FUNCTION_BLOCK "FB_ShuttleInt"   // FB57, SCL
{ S7_Optimized_Access := 'TRUE' }
// stored: MemoryReserve 100, SetENOAutomatically false
   VAR_INPUT
      iStartSeqCond : Bool;   // Start Sequence Conditions
      iJobReq : Bool;   // Job Request - From Main
      iIntGateOpened : Bool;   // Internal Gate Opened - From DI
      iIntGateClosed : Bool;   // Internal Gate Closed - From DI
      iExtGateOpened : Bool;   // External Gate Opened - From DI
      iExtGateClosed : Bool;   // External Gate Closed - From DI
      iShuttlePosInt : Bool;   // Shuttle Inside the Machine - Param
      iShuttlePosSas : Bool;   // Shuttle Inside the Sas - Param
      iShuttlePosExt : Bool;   // Shuttle Outside the Machine - Param
      iShuttlePosIntSetPoint : LReal;   // Shuttle Outside Position Setpoint - Param
      iShuttlePosSasSetPoint : LReal;   // Shuttle SasPosition Setpoint - Param
      iShuttleMoving : Bool;   // Shuttle is moving - From FB_LoaderAxis
      iShuttleInPos : Bool;   // Shuttle pos. reached - From FB_LoaderAxis
      iIntLoaderInSafePos : Bool;   // Gripper in Safe Position - Param
      iPLC_DateAndTime : DTL;
      iStepPause : Bool;
   END_VAR
   VAR_OUTPUT
      oExtGateOpenReq { ExternalAccessible := 'False'; ExternalVisible := 'False'; ExternalWritable := 'False'} : Bool;   // External Gate Opening Request - To DO
      oExtGateCloseReq { ExternalAccessible := 'False'; ExternalVisible := 'False'; ExternalWritable := 'False'} : Bool;   // External Gate Closing Request - To DO
      oIntGateOpenReq { ExternalAccessible := 'False'; ExternalVisible := 'False'; ExternalWritable := 'False'} : Bool;   // Internal Gate Opening Request - To DO
      oIntGateCloseReq { ExternalAccessible := 'False'; ExternalVisible := 'False'; ExternalWritable := 'False'} : Bool;   // Internal Gate Closing Request - To DO
      oShuttleStartReq { ExternalAccessible := 'False'; ExternalVisible := 'False'; ExternalWritable := 'False'} : Bool;   // Shuttle Start Order - To FB_LoaderAxis
      oShuttlePosSetPoint { ExternalAccessible := 'False'; ExternalVisible := 'False'; ExternalWritable := 'False'} : Real;   // Shuttle Position Setpoint - To FB_LoaderAxis
   END_VAR
   VAR
      sCurrent_Step_NB : Int;   // Active Step Number
      sCheck_Step_Condition : Bool;   // Check Step Condition
      sOneStepForward : Bool;
      sRTOneStepForward : R_TRIG;
      sOneStepMode { S7_SetPoint := 'True'} : Bool;
      sStepForward : Bool;
      sInterface : "UDT_SequenceInterface";   // Sequence Interface
      sExtGateOpenReq { ExternalAccessible := 'False'; ExternalVisible := 'False'; ExternalWritable := 'False'} : Bool;   // External Gate Opening Request
      sExtGateCloseReq { ExternalAccessible := 'False'; ExternalVisible := 'False'; ExternalWritable := 'False'} : Bool;   // External Gate Closing Request
      sIntGateOpenReq { ExternalAccessible := 'False'; ExternalVisible := 'False'; ExternalWritable := 'False'} : Bool;   // Internal Gate Opening Request
      sIntGateCloseReq { ExternalAccessible := 'False'; ExternalVisible := 'False'; ExternalWritable := 'False'} : Bool;   // Internal Gate Closing Request
      sShuttleStartReq { ExternalAccessible := 'False'; ExternalVisible := 'False'; ExternalWritable := 'False'} : Bool;   // Shuttle Start Request
      sShuttlePosSetPoint { ExternalAccessible := 'False'; ExternalVisible := 'False'; ExternalWritable := 'False'} : Real;   // Shuttle Position Setpoint
      sHistory : Struct
         Activation : Bool;
         Steps : Array[0..99] of Int;
         Date_Time : Array[0..99] of DTL;
      END_STRUCT;
      StepText : "FB_GetTextErrorCode";
   END_VAR
   VAR_TEMP
      tIndex : Int;   // Index
   END_VAR
   VAR CONSTANT
      S00_INIT : Int := 0;
      S10_CHECK_SHUTTLE_POSITION : Int := 10;
      S20_CLOSE_INT_GATE : Int := 20;
      S30_OPEN_EXT_GATE : Int := 30;
      S40_SHUTTLE_TO_SAS_START_REQ : Int := 40;
      S50_SHUTTLE_TO_SAS_POS_REACHED : Int := 50;
      S60_CLOSE_EXT_GATE : Int := 60;
      S70_OPEN_INT_GATE : Int := 70;
      S80_MOVE_SHUTTLE_TO_IN_START_REQ : Int := 80;
      S90_MOVE_SHUTTLE_TO_IN_POS_REACHED : Int := 90;
      S100_CLOSE_INT_GATE : Int := 100;
      S195_JOB_DONE : Int := 195;
   END_VAR
   // StepText.sCode_error[0].ErrorCode := 0;
   // StepText.sCode_error[1].ErrorCode := 10;
   // StepText.sCode_error[2].ErrorCode := 20;
   // StepText.sCode_error[3].ErrorCode := 30;
   // StepText.sCode_error[4].ErrorCode := 40;
   // StepText.sCode_error[5].ErrorCode := 50;
   // StepText.sCode_error[6].ErrorCode := 60;
   // StepText.sCode_error[7].ErrorCode := 70;
   // StepText.sCode_error[8].ErrorCode := 80;
   // StepText.sCode_error[9].ErrorCode := 90;
   // StepText.sCode_error[10].ErrorCode := 95;
   // StepText.sCode_error[0].ErrorText := 'S00 : INIT';
   // StepText.sCode_error[1].ErrorText := 'S10 : CHECK SHUTTLE POSITION';
   // StepText.sCode_error[2].ErrorText := 'S20 : OPEN EXT GATE';
   // StepText.sCode_error[3].ErrorText := 'S30 : SHUTTLE TO SAS START REQ';
   // StepText.sCode_error[4].ErrorText := 'S40 : SHUTTLE TO SAS POS REACHED';
   // StepText.sCode_error[5].ErrorText := 'S50 : CLOSE EXT GATE';
   // StepText.sCode_error[6].ErrorText := 'S60 : OPEN INT GATE';
   // StepText.sCode_error[7].ErrorText := 'S70 : MOVE SHUTTLE TO IN START REQ';
   // StepText.sCode_error[8].ErrorText := 'S80 : MOVE SHUTTLE TO IN POS REACHED';
   // StepText.sCode_error[9].ErrorText := 'S90 : CLOSE INT GATE';
   // StepText.sCode_error[10].ErrorText := 'S95 : JOB DONE';
BEGIN
   REGION Description header 
       //==================================================================================
       // POSALUX Swiss SA / (C) Copyright 2025
       //----------------------------------------------------------------------------------
       // Title: FB_ShuttleInt
       // Comment/Function: 
       // Author: Fabien WALDT
       // Engineering: TIA Portal v17
       //----------------------------------------------------------------------------------
       // Change log table:
       // Version  | Date     | Expert in charge | Changes applied
       // ---------|----------|------------------|-----------------------------------------
       // 00.00.01 | 20250527 | WFA              | First released version
       // =================================================================================
   END_REGION

   REGION Define condition to start
       IF #iStartSeqCond THEN
           #sInterface.SequenceReleased := TRUE;
       ELSE
           // Standard sequencer controls
           #sInterface.SequenceReleased := FALSE;
           #sCurrent_Step_NB := #S00_INIT;
           #sInterface.SequenceRun := FALSE;
           #sInterface.JobDone := FALSE;
           #sCheck_Step_Condition := FALSE;

           // Dedicated sequencer controls
           #sExtGateOpenReq := FALSE;
           #sExtGateCloseReq := FALSE;
           #sIntGateOpenReq := FALSE;
           #sIntGateCloseReq := FALSE;
           #sShuttleStartReq := FALSE;
           #sShuttlePosSetPoint := 0.0;
           // Add specifics controls 
       END_IF;

       // Reset interface error
       IF #sInterface.Reset THEN
           #sInterface.Error := FALSE;
       END_IF;

       // Reset start when axis in position
       IF #iShuttleInPos THEN
           #sShuttleStartReq := FALSE;
       END_IF;

       // One step forward
       #sRTOneStepForward.CLK := #sOneStepForward;
       #sRTOneStepForward();
       #sStepForward := (NOT #sOneStepMode OR (#sOneStepMode AND #sRTOneStepForward.Q)) AND NOT #iStepPause;
       #sOneStepForward := FALSE;
   END_REGION

   REGION Sequence Function
       CASE #sCurrent_Step_NB OF
           #S00_INIT:
               REGION S00 INIT
                   #sCheck_Step_Condition := TRUE;
               END_REGION
           #S10_CHECK_SHUTTLE_POSITION:
               REGION S10_CHECK_SHUTTLE_POSITION
                   #sCheck_Step_Condition := TRUE;
               END_REGION
           #S20_CLOSE_INT_GATE:
               REGION S20_CLOSE_INT_GATE
                   #sIntGateOpenReq := FALSE;
                   #sIntGateCloseReq := TRUE;
                   #sCheck_Step_Condition := TRUE;
               END_REGION
           #S30_OPEN_EXT_GATE:
               REGION S30_OPEN_EXT_GATE
                   #sExtGateOpenReq := TRUE;
                   #sExtGateCloseReq := FALSE;
                   #sCheck_Step_Condition := TRUE;
               END_REGION
           #S40_SHUTTLE_TO_SAS_START_REQ:
               REGION S40_SHUTTLE_TO_SAS_START_REQ
                   #sShuttleStartReq := #iExtGateOpened AND NOT #iShuttlePosSas;
                   #sShuttlePosSetPoint := LREAL_TO_REAL(#iShuttlePosSasSetPoint);
                   #sCheck_Step_Condition := TRUE;
               END_REGION
           #S50_SHUTTLE_TO_SAS_POS_REACHED:
               REGION S50_SHUTTLE_TO_SAS_POS_REACHED
                   #sCheck_Step_Condition := TRUE;
               END_REGION
           #S60_CLOSE_EXT_GATE:
               REGION S60_CLOSE_EXT_GATE
                   #sExtGateOpenReq := FALSE;
                   #sExtGateCloseReq := TRUE;
                   #sCheck_Step_Condition := TRUE;
               END_REGION
           #S70_OPEN_INT_GATE:
               REGION S70_OPEN_INT_GATE
                   #sIntGateOpenReq := TRUE;
                   #sIntGateCloseReq := FALSE;
                   #sCheck_Step_Condition := TRUE;
               END_REGION
           #S80_MOVE_SHUTTLE_TO_IN_START_REQ:
               REGION S80_MOVE_SHUTTLE_TO_IN_START_REQ
                   #sShuttleStartReq := #iIntGateOpened AND NOT #iShuttlePosInt;
                   #sShuttlePosSetPoint := LREAL_TO_REAL(#iShuttlePosIntSetPoint);
                   #sCheck_Step_Condition := TRUE;
               END_REGION
           #S90_MOVE_SHUTTLE_TO_IN_POS_REACHED:
               REGION S90_MOVE_SHUTTLE_TO_IN_POS_REACHED
                   #sCheck_Step_Condition := TRUE;
               END_REGION
           #S100_CLOSE_INT_GATE:
               REGION S100_CLOSE_INT_GATE
                   #sIntGateOpenReq := FALSE;
                   #sIntGateCloseReq := TRUE;
                   #sExtGateOpenReq := FALSE;
                   #sExtGateCloseReq := TRUE;
                   #sCheck_Step_Condition := TRUE;
               END_REGION
           #S195_JOB_DONE:
               REGION S195_JOB_DONE
                   #sInterface.JobDone := TRUE;
                   #sCheck_Step_Condition := TRUE;
               END_REGION
           ELSE:
               #sInterface.Error := TRUE;
       END_CASE;
   END_REGION

   REGION Sequence Next Step Condition
       IF #sCheck_Step_Condition THEN
           CASE #sCurrent_Step_NB OF
               #S00_INIT:
                   REGION S00 INIT
                       IF #sInterface.SequenceReleased AND #iJobReq THEN
                           #sCurrent_Step_NB := #S10_CHECK_SHUTTLE_POSITION;
                           #sInterface.SequenceRun := TRUE;
                           #sCheck_Step_Condition := FALSE;
                       ELSE
                           #sInterface.SequenceRun := FALSE;
                       END_IF;
                   END_REGION
               #S10_CHECK_SHUTTLE_POSITION:
                   REGION S10_CHECK_SHUTTLE_POSITION
                       IF #sInterface.SequenceReleased AND #sStepForward AND #iShuttlePosExt THEN
                           #sCurrent_Step_NB := #S20_CLOSE_INT_GATE;
                           #sCheck_Step_Condition := FALSE;
                       ELSIF #sInterface.SequenceReleased AND #sStepForward AND #iShuttlePosSas THEN
                           #sCurrent_Step_NB := #S60_CLOSE_EXT_GATE;
                           #sCheck_Step_Condition := FALSE;
                       ELSIF #sInterface.SequenceReleased AND #sStepForward AND #iShuttlePosInt THEN
                           #sCurrent_Step_NB := #S100_CLOSE_INT_GATE;
                           #sCheck_Step_Condition := FALSE;
                       END_IF;
                   END_REGION
               #S20_CLOSE_INT_GATE:
                   REGION S20_CLOSE_INT_GATE
                       IF #sInterface.SequenceReleased AND #sStepForward AND #iIntGateClosed THEN
                           #sCurrent_Step_NB := #S30_OPEN_EXT_GATE;
                           #sCheck_Step_Condition := FALSE;
                       END_IF;
                   END_REGION
               #S30_OPEN_EXT_GATE:
                   REGION S30_OPEN_EXT_GATE
                       IF #sInterface.SequenceReleased AND #sStepForward AND #iExtGateOpened THEN
                           #sCurrent_Step_NB := #S40_SHUTTLE_TO_SAS_START_REQ;
                           #sCheck_Step_Condition := FALSE;
                       END_IF;
                   END_REGION
               #S40_SHUTTLE_TO_SAS_START_REQ:
                   REGION S40_SHUTTLE_TO_SAS_START_REQ
                      // IF #sInterface.SequenceReleased AND #sStepForward AND (#ShuttleMoving OR #ShuttlePosSas)  THEN
                       IF #sInterface.SequenceReleased AND (#iShuttleMoving OR #iShuttlePosSas)  THEN
                           #sCurrent_Step_NB := #S50_SHUTTLE_TO_SAS_POS_REACHED;
                           #sCheck_Step_Condition := FALSE;
                       END_IF;
                   END_REGION
               #S50_SHUTTLE_TO_SAS_POS_REACHED:
                   REGION S50_SHUTTLE_TO_SAS_POS_REACHED
                       IF #sInterface.SequenceReleased AND #sStepForward AND NOT #sShuttleStartReq AND #iShuttlePosSas THEN
                           #sCurrent_Step_NB := #S60_CLOSE_EXT_GATE;
                           #sCheck_Step_Condition := FALSE;
                       END_IF;
                   END_REGION
               #S60_CLOSE_EXT_GATE:
                   REGION S60_CLOSE_EXT_GATE
                       IF #sInterface.SequenceReleased AND #sStepForward AND #iExtGateClosed THEN
                           #sCurrent_Step_NB := #S70_OPEN_INT_GATE;
                           #sCheck_Step_Condition := FALSE;
                       END_IF;
                   END_REGION
               #S70_OPEN_INT_GATE:
                   REGION S70_OPEN_INT_GATE
                       IF #sInterface.SequenceReleased AND #sStepForward AND #iIntGateOpened THEN
                           #sCurrent_Step_NB := #S80_MOVE_SHUTTLE_TO_IN_START_REQ;
                           #sCheck_Step_Condition := FALSE;
                       END_IF;
                   END_REGION
               #S80_MOVE_SHUTTLE_TO_IN_START_REQ:
                   REGION S80_MOVE_SHUTTLE_TO_IN_START_REQ
                       IF #sInterface.SequenceReleased AND (#iShuttleMoving OR #iShuttlePosInt) THEN
                           #sCurrent_Step_NB := #S90_MOVE_SHUTTLE_TO_IN_POS_REACHED;
                           #sCheck_Step_Condition := FALSE;
                       END_IF;
                   END_REGION
               #S90_MOVE_SHUTTLE_TO_IN_POS_REACHED:
                   REGION S90_MOVE_SHUTTLE_TO_IN_POS_REACHED
                       IF #sInterface.SequenceReleased AND #sStepForward AND NOT #sShuttleStartReq AND #iShuttlePosInt THEN
                           #sCurrent_Step_NB := #S100_CLOSE_INT_GATE;
                           #sCheck_Step_Condition := FALSE;
                       END_IF;
                   END_REGION
               #S100_CLOSE_INT_GATE:
                   REGION S100_CLOSE_INT_GATE
                       IF #sInterface.SequenceReleased AND #sStepForward AND #iIntGateClosed AND #iExtGateClosed THEN
                           #sCurrent_Step_NB := #S195_JOB_DONE;
                           #sCheck_Step_Condition := FALSE;
                       END_IF;
                   END_REGION
               #S195_JOB_DONE:
                   REGION S195_JOB_DONE
                       IF NOT #iJobReq THEN
                           #sCurrent_Step_NB := #S00_INIT;
                           #sCheck_Step_Condition := FALSE;
                           #sInterface.JobDone := FALSE;
                       END_IF;
                   END_REGION
               ELSE
                   #sInterface.Error := TRUE;
           END_CASE;
       END_IF;
   END_REGION

   REGION Outputs Update
       #oExtGateOpenReq  := #sExtGateOpenReq;
       #oExtGateCloseReq := #sExtGateCloseReq;
       #oIntGateOpenReq  := #sIntGateOpenReq;
       #oIntGateCloseReq := #sIntGateCloseReq;
       #oShuttleStartReq := #sShuttleStartReq AND ((#iShuttlePosInt AND #iIntLoaderInSafePos) OR NOT #iShuttlePosInt);
       #oShuttlePosSetPoint:= #sShuttlePosSetPoint;
   END_REGION

   REGION Steps - Date and Time History
       IF #sHistory.Activation THEN
           IF #sHistory.Steps[0] <> #sCurrent_Step_NB THEN
               FOR #tIndex := 98 TO 0 BY -1 DO
                   #sHistory.Steps[#tIndex + 1] := #sHistory.Steps[#tIndex];
                   #sHistory.Date_Time[#tIndex + 1] := #sHistory.Date_Time[#tIndex];
               END_FOR;
               #sHistory.Steps[0] := #sCurrent_Step_NB;
               #sHistory.Date_Time[0] := #iPLC_DateAndTime;
           END_IF;
       END_IF;
   END_REGION

   REGION Steps Text
       #StepText(iErrorCode:=#sCurrent_Step_NB,
                 oErrorText=>#StepText.oErrorText);
   END_REGION
END_FUNCTION_BLOCK

FUNCTION_BLOCK "FB_ShuttleExt"   // FB59, SCL
{ S7_Optimized_Access := 'TRUE' }
// stored: MemoryReserve 100, SetENOAutomatically false
   VAR_INPUT
      iStartSeqCond : Bool;   // Start Sequence Conditions
      iJobReq : Bool;   // Job Request - From Main
      iIntGateOpened : Bool;   // Internal Gate Opened - From DI
      iIntGateClosed : Bool;   // Internal Gate Closed - From DI
      iExtGateOpened : Bool;   // External Gate Opened - From DI
      iExtGateClosed : Bool;   // External Gate Closed - From DI
      iShuttlePosInt : Bool;   // Shuttle Inside the Machine - Param
      iShuttlePosSas : Bool;   // Shuttle Inside the Sas - Param
      iShuttlePosExt : Bool;   // Shuttle Outside the Machine - Param
      iShuttlePosExtSetPoint : LReal;   // Shuttle Outside Position Setpoint - Param
      iShuttlePosSasSetPoint : LReal;   // Shuttle SasPosition Setpoint - Param
      iShuttleMoving : Bool;   // Shuttle is moving - From FB_LoaderAxis
      iShuttleInPos : Bool;   // Shuttle pos. reached - From FB_LoaderAxis
      iExtLoaderInSafePos : Bool;   // Gripper in Safe Position - Param
      iPLC_DateAndTime : DTL;
      iStepPause : Bool;
   END_VAR
   VAR_OUTPUT
      oExtGateOpenReq { ExternalAccessible := 'False'; ExternalVisible := 'False'; ExternalWritable := 'False'} : Bool;   // External Gate Opening Request - To DO
      oExtGateCloseReq { ExternalAccessible := 'False'; ExternalVisible := 'False'; ExternalWritable := 'False'} : Bool;   // External Gate Closing Request - To DO
      oIntGateOpenReq { ExternalAccessible := 'False'; ExternalVisible := 'False'; ExternalWritable := 'False'} : Bool;   // Internal Gate Opening Request - To DO
      oIntGateCloseReq { ExternalAccessible := 'False'; ExternalVisible := 'False'; ExternalWritable := 'False'} : Bool;   // Internal Gate Closing Request - To DO
      oShuttleStartReq { ExternalAccessible := 'False'; ExternalVisible := 'False'; ExternalWritable := 'False'} : Bool;   // Shuttle Start Order - To FB_LoaderAxis
      oShuttlePosSetPoint { ExternalAccessible := 'False'; ExternalVisible := 'False'; ExternalWritable := 'False'} : Real;   // Shuttle Position Setpoint - To FB_LoaderAxis
   END_VAR
   VAR
      sCurrent_Step_NB : Int;   // Active Step Number
      sCheck_Step_Condition : Bool;   // Check Step Condition
      sOneStepForward : Bool;
      sRTOneStepForward : R_TRIG;
      sOneStepMode { S7_SetPoint := 'True'} : Bool;
      sStepForward : Bool;
      sInterface : "UDT_SequenceInterface";   // Sequence Interface
      sExtGateOpenReq { ExternalAccessible := 'False'; ExternalVisible := 'False'; ExternalWritable := 'False'} : Bool;   // External Gate Opening Request
      sExtGateCloseReq { ExternalAccessible := 'False'; ExternalVisible := 'False'; ExternalWritable := 'False'} : Bool;   // External Gate Closing Request
      sIntGateOpenReq { ExternalAccessible := 'False'; ExternalVisible := 'False'; ExternalWritable := 'False'} : Bool;   // Internal Gate Opening Request
      sIntGateCloseReq { ExternalAccessible := 'False'; ExternalVisible := 'False'; ExternalWritable := 'False'} : Bool;   // Internal Gate Closing Request
      sShuttleStartReq { ExternalAccessible := 'False'; ExternalVisible := 'False'; ExternalWritable := 'False'} : Bool;   // Shuttle Start Request
      sShuttlePosSetPoint { ExternalAccessible := 'False'; ExternalVisible := 'False'; ExternalWritable := 'False'} : Real;   // Shuttle Position Setpoint
      sHistory : Struct
         Activation : Bool;
         Steps : Array[0..99] of Int;
         Date_Time : Array[0..99] of DTL;
      END_STRUCT;
      StepText : "FB_GetTextErrorCode";
   END_VAR
   VAR_TEMP
      tIndex : Int;   // Index
   END_VAR
   VAR CONSTANT
      S00_INIT : Int := 0;
      S10_CHECK_SHUTTLE_POSITION : Int := 10;
      S20_CLOSE_EXT_GATE : Int := 20;
      S30_OPEN_INT_GATE : Int := 30;
      S40_SHUTTLE_TO_SAS_START_REQ : Int := 40;
      S50_SHUTTLE_TO_SAS_POS_REACHED : Int := 50;
      S60_CLOSE_INT_GATE : Int := 60;
      S70_OPEN_EXT_GATE : Int := 70;
      S80_MOVE_SHUTTLE_TO_OUT_START_REQ : Int := 80;
      S90_MOVE_SHUTTLE_TO_OUT_POS_REACHED : Int := 90;
      S100_CLOSE_EXT_GATE : Int := 100;
      S195_JOB_DONE : Int := 195;
   END_VAR
   // StepText.sCode_error[0].ErrorCode := 0;
   // StepText.sCode_error[1].ErrorCode := 10;
   // StepText.sCode_error[2].ErrorCode := 20;
   // StepText.sCode_error[3].ErrorCode := 30;
   // StepText.sCode_error[4].ErrorCode := 40;
   // StepText.sCode_error[5].ErrorCode := 50;
   // StepText.sCode_error[6].ErrorCode := 60;
   // StepText.sCode_error[7].ErrorCode := 70;
   // StepText.sCode_error[8].ErrorCode := 80;
   // StepText.sCode_error[9].ErrorCode := 90;
   // StepText.sCode_error[10].ErrorCode := 95;
   // StepText.sCode_error[0].ErrorText := 'S00 : INIT';
   // StepText.sCode_error[1].ErrorText := 'S10 : CHECK SHUTTLE POSITION';
   // StepText.sCode_error[2].ErrorText := 'S20 : OPEN INT GATE';
   // StepText.sCode_error[3].ErrorText := 'S30 : SHUTTLE TO SAS START REQ';
   // StepText.sCode_error[4].ErrorText := 'S40 : SHUTTLE TO SAS POS REACHED';
   // StepText.sCode_error[5].ErrorText := 'S50 : CLOSE INT GATE';
   // StepText.sCode_error[6].ErrorText := 'S60 : OPEN EXT GATE';
   // StepText.sCode_error[7].ErrorText := 'S70 : MOVE SHUTTLE TO OUT START REQ';
   // StepText.sCode_error[8].ErrorText := 'S80 : MOVE SHUTTLE TO OUT POS REACHED';
   // StepText.sCode_error[9].ErrorText := 'S90 : CLOSE EXT GATE';
   // StepText.sCode_error[10].ErrorText := 'S95 : JOB DONE';
BEGIN
   REGION Description header 
       //==================================================================================
       // POSALUX Swiss SA / (C) Copyright 2025
       //----------------------------------------------------------------------------------
       // Title: FB_ShuttleExt
       // Comment/Function: 
       // Author: Fabien WALDT
       // Engineering: TIA Portal v17
       //----------------------------------------------------------------------------------
       // Change log table:
       // Version  | Date     | Expert in charge | Changes applied
       // ---------|----------|------------------|-----------------------------------------
       // 00.00.01 | 20250527 | WFA              | First released version
       // =================================================================================
   END_REGION

   REGION Define condition to start
       IF #iStartSeqCond THEN
           #sInterface.SequenceReleased := TRUE;
       ELSE
           // Standard sequencer controls
           #sInterface.SequenceReleased := FALSE;
           #sCurrent_Step_NB := #S00_INIT;
           #sInterface.SequenceRun := FALSE;
           #sInterface.JobDone := FALSE;
           #sCheck_Step_Condition := FALSE;

           // Dedicated sequencer controls
           #sExtGateOpenReq := FALSE;
           #sExtGateCloseReq := FALSE;
           #sIntGateOpenReq := FALSE;
           #sIntGateCloseReq := FALSE;
           #sShuttleStartReq := FALSE;
           #sShuttlePosSetPoint := 0.0;
           // Add specifics controls 
       END_IF;

       // Reset interface error
       IF #sInterface.Reset THEN
           #sInterface.Error := FALSE;
       END_IF;

       // Reset start when axis in position
       IF #iShuttleInPos THEN
           #sShuttleStartReq := FALSE;
       END_IF;

       // One step forward
       #sRTOneStepForward.CLK := #sOneStepForward;
       #sRTOneStepForward();
       #sStepForward := (NOT #sOneStepMode OR (#sOneStepMode AND #sRTOneStepForward.Q)) AND NOT #iStepPause;
       #sOneStepForward := FALSE;
   END_REGION

   REGION Sequence Function
       CASE #sCurrent_Step_NB OF
           #S00_INIT:
               REGION S00 INIT
                   #sCheck_Step_Condition := TRUE;
               END_REGION
           #S10_CHECK_SHUTTLE_POSITION:
               REGION S10_CHECK_SHUTTLE_POSITION
                   #sCheck_Step_Condition := TRUE;
               END_REGION
           #S20_CLOSE_EXT_GATE:
               REGION S20_CLOSE_EXT_GATE
                   #sExtGateOpenReq := FALSE;
                   #sExtGateCloseReq := TRUE;
                   #sCheck_Step_Condition := TRUE;
               END_REGION
           #S30_OPEN_INT_GATE:
               REGION S30_OPEN_INT_GATE
                   #sIntGateOpenReq := TRUE;
                   #sIntGateCloseReq := FALSE;
                   #sCheck_Step_Condition := TRUE;
               END_REGION
           #S40_SHUTTLE_TO_SAS_START_REQ:
               REGION S40_SHUTTLE_TO_SAS_START_REQ
                   #sShuttleStartReq := #iIntGateOpened AND NOT #iShuttlePosSas;
                   #sShuttlePosSetPoint := LREAL_TO_REAL(#iShuttlePosSasSetPoint);
                   #sCheck_Step_Condition := TRUE;
               END_REGION
           #S50_SHUTTLE_TO_SAS_POS_REACHED:
               REGION S50_SHUTTLE_TO_SAS_POS_REACHED
                   #sCheck_Step_Condition := TRUE;
               END_REGION
           #S60_CLOSE_INT_GATE:
               REGION S60_CLOSE_INT_GATE
                   #sIntGateOpenReq := FALSE;
                   #sIntGateCloseReq := TRUE;
                   #sCheck_Step_Condition := TRUE;
               END_REGION
           #S70_OPEN_EXT_GATE:
               REGION S70_OPEN_EXT_GATE
                   #sExtGateOpenReq := TRUE;
                   #sExtGateCloseReq := FALSE;
                   #sCheck_Step_Condition := TRUE;
               END_REGION
           #S80_MOVE_SHUTTLE_TO_OUT_START_REQ:
               REGION S80_MOVE_SHUTTLE_TO_OUT_START_REQ
                   #sShuttleStartReq := #iExtGateOpened AND NOT #iShuttlePosExt;
                   #sShuttlePosSetPoint := LREAL_TO_REAL(#iShuttlePosExtSetPoint);
                   #sCheck_Step_Condition := TRUE;
               END_REGION
           #S90_MOVE_SHUTTLE_TO_OUT_POS_REACHED:
               REGION S90_MOVE_SHUTTLE_TO_OUT_POS_REACHED
                   #sCheck_Step_Condition := TRUE;
               END_REGION
           #S100_CLOSE_EXT_GATE:
               REGION S100_CLOSE_EXT_GATE
                   #sIntGateOpenReq := FALSE;
                   #sIntGateCloseReq := TRUE;
                   #sExtGateOpenReq := FALSE;
                   #sExtGateCloseReq := TRUE;
                   #sCheck_Step_Condition := TRUE;
               END_REGION
           #S195_JOB_DONE:
               REGION S195_JOB_DONE
                   #sInterface.JobDone := TRUE;
                   #sCheck_Step_Condition := TRUE;
               END_REGION
           ELSE:
               #sInterface.Error := TRUE;
       END_CASE;
   END_REGION

   REGION Sequence Next Step Condition
       IF #sCheck_Step_Condition THEN
           CASE #sCurrent_Step_NB OF
               #S00_INIT:
                   REGION S00 INIT
                       IF #sInterface.SequenceReleased AND #iJobReq THEN
                           #sCurrent_Step_NB := #S10_CHECK_SHUTTLE_POSITION;
                           #sInterface.SequenceRun := TRUE;
                           #sCheck_Step_Condition := FALSE;
                       ELSE
                           #sInterface.SequenceRun := FALSE;
                       END_IF;
                   END_REGION
               #S10_CHECK_SHUTTLE_POSITION:
                   REGION S10_CHECK_SHUTTLE_POSITION
                       IF #sInterface.SequenceReleased AND #sStepForward AND #iShuttlePosInt THEN
                           #sCurrent_Step_NB := #S20_CLOSE_EXT_GATE;
                           #sCheck_Step_Condition := FALSE;
                       ELSIF #sInterface.SequenceReleased AND #sStepForward AND #iShuttlePosSas THEN
                           #sCurrent_Step_NB := #S60_CLOSE_INT_GATE;
                           #sCheck_Step_Condition := FALSE;
                       ELSIF #sInterface.SequenceReleased AND #sStepForward AND #iShuttlePosExt THEN
                           #sCurrent_Step_NB := #S100_CLOSE_EXT_GATE;
                           #sCheck_Step_Condition := FALSE;
                       END_IF;
                   END_REGION
               #S20_CLOSE_EXT_GATE:
                   REGION S20_CLOSE_EXT_GATE
                       IF #sInterface.SequenceReleased AND #sStepForward AND #iExtGateClosed THEN
                           #sCurrent_Step_NB := #S30_OPEN_INT_GATE;
                           #sCheck_Step_Condition := FALSE;
                       END_IF;
                   END_REGION
               #S30_OPEN_INT_GATE:
                   REGION S30_OPEN_INT_GATE
                       IF #sInterface.SequenceReleased AND #sStepForward AND #iIntGateOpened THEN
                           #sCurrent_Step_NB := #S40_SHUTTLE_TO_SAS_START_REQ;
                           #sCheck_Step_Condition := FALSE;
                       END_IF;
                   END_REGION
               #S40_SHUTTLE_TO_SAS_START_REQ:
                   REGION S40_SHUTTLE_TO_SAS_START_REQ
                     //  IF #sInterface.SequenceReleased AND #sStepForward AND (#ShuttleMoving OR #ShuttlePosSas) THEN
                       IF #sInterface.SequenceReleased AND (#iShuttleMoving OR #iShuttlePosSas) THEN
                           #sCurrent_Step_NB := #S50_SHUTTLE_TO_SAS_POS_REACHED;
                           #sCheck_Step_Condition := FALSE;
                       END_IF;
                   END_REGION
               #S50_SHUTTLE_TO_SAS_POS_REACHED:
                   REGION S50_SHUTTLE_TO_SAS_POS_REACHED
                       IF #sInterface.SequenceReleased AND #sStepForward AND NOT #sShuttleStartReq AND #iShuttlePosSas THEN
                           #sCurrent_Step_NB := #S60_CLOSE_INT_GATE;
                           #sCheck_Step_Condition := FALSE;
                       END_IF;
                   END_REGION
               #S60_CLOSE_INT_GATE:
                   REGION S60_CLOSE_INT_GATE
                       IF #sInterface.SequenceReleased AND #sStepForward AND #iIntGateClosed THEN
                           #sCurrent_Step_NB := #S70_OPEN_EXT_GATE;
                           #sCheck_Step_Condition := FALSE;
                       END_IF;
                   END_REGION
               #S70_OPEN_EXT_GATE:
                   REGION S70_OPEN_EXT_GATE
                       IF #sInterface.SequenceReleased AND #sStepForward AND #iExtGateOpened THEN
                           #sCurrent_Step_NB := #S80_MOVE_SHUTTLE_TO_OUT_START_REQ;
                           #sCheck_Step_Condition := FALSE;
                       END_IF;
                   END_REGION
               #S80_MOVE_SHUTTLE_TO_OUT_START_REQ:
                   REGION S80_MOVE_SHUTTLE_TO_OUT_START_REQ
                       IF #sInterface.SequenceReleased AND (#iShuttleMoving OR #iShuttlePosExt) THEN
                           #sCurrent_Step_NB := #S90_MOVE_SHUTTLE_TO_OUT_POS_REACHED;
                           #sCheck_Step_Condition := FALSE;
                       END_IF;
                   END_REGION
               #S90_MOVE_SHUTTLE_TO_OUT_POS_REACHED:
                   REGION S90_MOVE_SHUTTLE_TO_OUT_POS_REACHED
                       IF #sInterface.SequenceReleased AND #sStepForward AND NOT #sShuttleStartReq AND #iShuttlePosExt THEN
                           #sCurrent_Step_NB := #S100_CLOSE_EXT_GATE;
                           #sCheck_Step_Condition := FALSE;
                       END_IF;
                   END_REGION
               #S100_CLOSE_EXT_GATE:
                   REGION S100_CLOSE_EXT_GATE
                       IF #sInterface.SequenceReleased AND #sStepForward AND #iIntGateClosed AND #iExtGateClosed THEN
                           #sCurrent_Step_NB := #S195_JOB_DONE;
                           #sCheck_Step_Condition := FALSE;
                       END_IF;
                   END_REGION
               #S195_JOB_DONE:
                   REGION S195_JOB_DONE
                       IF NOT #iJobReq THEN
                           #sCurrent_Step_NB := #S00_INIT;
                           #sCheck_Step_Condition := FALSE;
                           #sInterface.JobDone := FALSE;
                       END_IF;
                   END_REGION
               ELSE
                   #sInterface.Error := TRUE;
           END_CASE;
       END_IF;
   END_REGION

   REGION Outputs Update
       #oExtGateOpenReq  := #sExtGateOpenReq;
       #oExtGateCloseReq := #sExtGateCloseReq;
       #oIntGateOpenReq  := #sIntGateOpenReq;
       #oIntGateCloseReq := #sIntGateCloseReq;
       #oShuttleStartReq:= #sShuttleStartReq AND ((#iShuttlePosExt AND #iExtLoaderInSafePos) OR NOT #iShuttlePosExt);
       #oShuttlePosSetPoint:= #sShuttlePosSetPoint;
   END_REGION

   REGION Steps - Date and Time History
       IF #sHistory.Activation THEN
           IF #sHistory.Steps[0] <> #sCurrent_Step_NB THEN
               FOR #tIndex := 98 TO 0 BY -1 DO
                   #sHistory.Steps[#tIndex + 1] := #sHistory.Steps[#tIndex];
                   #sHistory.Date_Time[#tIndex + 1] := #sHistory.Date_Time[#tIndex];
               END_FOR;
               #sHistory.Steps[0] := #sCurrent_Step_NB;
               #sHistory.Date_Time[0] := #iPLC_DateAndTime;
           END_IF;
       END_IF;
   END_REGION

   REGION Steps Text
       #StepText(iErrorCode := #sCurrent_Step_NB,
                 oErrorText => #StepText.oErrorText);
   END_REGION
END_FUNCTION_BLOCK

FUNCTION_BLOCK "FB_ExtLoadUnload"   // FB61, SCL
{ S7_Optimized_Access := 'TRUE' }
// stored: MemoryReserve 100, SetENOAutomatically false
   VAR_INPUT
      iStartSeqCond : Bool;   // Start Sequence Conditions
      iJobReq : Bool;   // Job Request - From Main
      iShuttleExtLoadUnloadAutoPos : Bool;   // Load/Unload Auto Pos. Reached - Param
      iShuttleExtLoadUnloadAutoPosSetPoint : LReal;   // Load/Unload Auto Pos. Setpoint - Param
      iShuttleExtLoadUnloadManuPos : Bool;   // Load/Unload Manu Pos. Reached - Param
      iShuttleExtLoadUnloadManuPosSetPoint : LReal;   // Load/Unload Manu Pos. Setpoint - Param
      iShuttleMoving : Bool;   // Shuttle is moving - From FB_LoaderAxis
      iShuttleInPos : Bool;   // Shuttle pos. reached - From FB_LoaderAxis
      iCommunicationWithExtLoaderDone : Bool;   // Communication Done - From Ext Loader
      iLoadUnloadMsgManuModeAck : Bool;   // Load/Unload Message Ack - From HMI
      iAutoMode : Bool;
      iSemiAutoMode : Bool;
      iFillingMode : Bool;   // Filling Mode - From Machine States
      iEmptyingMode : Bool;   // Emptying Mode - From Machine States
      iPLC_DateAndTime : DTL;
      iStepPause : Bool;
   END_VAR
   VAR_OUTPUT
      oShuttleStartReq { ExternalAccessible := 'False'; ExternalVisible := 'False'; ExternalWritable := 'False'} : Bool;   // Shuttle Start Order - To FB_LoaderAxis
      oShuttlePosSetPoint { ExternalAccessible := 'False'; ExternalVisible := 'False'; ExternalWritable := 'False'} : Real;   // Shuttle Position Setpoint - To FB_LoaderAxis
      oStartCommunicationWithExtLoader : Bool;   // Start Communication - To Ext Loader
      oSetLoadUnloadMsgManuMode : Bool;   // Set Load/Unload Message - To HMI
   END_VAR
   VAR
      sCurrent_Step_NB : Int;   // Active Step Number
      sCheck_Step_Condition : Bool;
      sOneStepForward : Bool;
      sRTOneStepForward : R_TRIG;
      sOneStepMode { S7_SetPoint := 'True'} : Bool;
      sStepForward : Bool;
      sInterface : "UDT_SequenceInterface";
      sShuttleStartReq { ExternalAccessible := 'False'; ExternalVisible := 'False'; ExternalWritable := 'False'} : Bool;
      sShuttlePosSetPoint { ExternalAccessible := 'False'; ExternalVisible := 'False'; ExternalWritable := 'False'} : Real;
      sHistory : Struct
         Activation : Bool;
         Steps : Array[0..99] of Int;
         Date_Time : Array[0..99] of DTL;
      END_STRUCT;
      StepText : "FB_GetTextErrorCode";
   END_VAR
   VAR_TEMP
      tIndex : Int;   // Index
   END_VAR
   VAR CONSTANT
      S00_INIT : Int := 0;
      S10_CHECK_EXT_LOAD_UNLOAD_OPTION : Int := 10;
      S20_SHUTTLE_TO_EXT_LOAD_UNLOAD_POS_START_REQ : Int := 20;
      S30_SHUTTLE_TO_EXT_LOAD_UNLOAD_POS_REACHED : Int := 30;
      S40_SET_EXCHANGE_EXT_LOADER_LOAD_UNLOAD : Int := 40;
      S50_EXCHANGE_EXT_LOADER_IN_PROGRESS : Int := 50;
      S60_EXCHANGE_EXT_LOADER_ACQUIT : Int := 60;
      S70_SET_EXCHANGE_EXT_LOADER_UNLOAD : Int := 70;
      S80_EXCHANGE_EXT_LOADER_IN_PROGRESS : Int := 80;
      S90_EXCHANGE_EXT_LOADER_ACQUIT : Int := 90;
      S100_SET_EXCHANGE_EXT_LOADER_UNLOAD : Int := 100;
      S110_EXCHANGE_EXT_LOADER_IN_PROGRESS : Int := 110;
      S120_EXCHANGE_EXT_LOADER_ACQUIT : Int := 120;
      S130_SHUTTLE_TO_EXT_LOAD_UNLOAD_MANU_POS_START_REQ : Int := 130;
      S140_SHUTTLE_TO_EXT_LOAD_UNLOAD_MANU_POS_REACHED : Int := 140;
      S150_OPERATOR_MESSAGE : Int := 150;
      S195_JOB_DONE : Int := 195;
   END_VAR
   // StepText.sCode_error[0].ErrorCode := 0;
   // StepText.sCode_error[1].ErrorCode := 10;
   // StepText.sCode_error[2].ErrorCode := 20;
   // StepText.sCode_error[3].ErrorCode := 30;
   // StepText.sCode_error[4].ErrorCode := 40;
   // StepText.sCode_error[5].ErrorCode := 50;
   // StepText.sCode_error[6].ErrorCode := 60;
   // StepText.sCode_error[7].ErrorCode := 70;
   // StepText.sCode_error[8].ErrorCode := 80;
   // StepText.sCode_error[9].ErrorCode := 90;
   // StepText.sCode_error[10].ErrorCode := 95;
BEGIN
   REGION Description header 
       //==================================================================================
       // POSALUX Swiss SA / (C) Copyright 2025
       //----------------------------------------------------------------------------------
       // Title: FB_ExtLoadUnload
       // Comment/Function: 
       // Author: Fabien WALDT
       // Engineering: TIA Portal v17
       //----------------------------------------------------------------------------------
       // Change log table:
       // Version  | Date     | Expert in charge | Changes applied
       // ---------|----------|------------------|-----------------------------------------
       // 00.00.01 | 20250527 | WFA              | First released version
       // =================================================================================
   END_REGION

   REGION Define condition to start
       IF #iStartSeqCond THEN
           #sInterface.SequenceReleased := TRUE;
       ELSE
           // Standard sequencer controls
           #sInterface.SequenceReleased := FALSE;
           #sCurrent_Step_NB := #S00_INIT;
           #sInterface.SequenceRun := FALSE;
           #sInterface.JobDone := FALSE;
           #sCheck_Step_Condition := FALSE;

           // Dedicated sequencer controls
           #sShuttleStartReq := FALSE;
           #sShuttlePosSetPoint := 0.0;
           #oStartCommunicationWithExtLoader := FALSE;
           // Add specifics controls 
       END_IF;

       // Reset interface error
       IF #sInterface.Reset THEN
           #sInterface.Error := FALSE;
       END_IF;

       // Reset start when axis in position
       IF #iShuttleInPos THEN
           #sShuttleStartReq := FALSE;
       END_IF;

       // One step forward
       #sRTOneStepForward.CLK := #sOneStepForward;
       #sRTOneStepForward();
       #sStepForward := (NOT #sOneStepMode OR (#sOneStepMode AND #sRTOneStepForward.Q)) AND NOT #iStepPause;
       #sOneStepForward := FALSE;

       // Action only true in dedicated steps
       #oSetLoadUnloadMsgManuMode := FALSE;
   END_REGION

   REGION Sequence Function
       CASE #sCurrent_Step_NB OF
           #S00_INIT:
               REGION S00 INIT
                   #sCheck_Step_Condition := TRUE;
               END_REGION
           #S10_CHECK_EXT_LOAD_UNLOAD_OPTION:
               REGION S10_CHECK_EXT_LOAD_UNLOAD_OPTION
                   #sCheck_Step_Condition := TRUE;
               END_REGION
           #S20_SHUTTLE_TO_EXT_LOAD_UNLOAD_POS_START_REQ:
               REGION S20_SHUTTLE_TO_EXT_LOAD_UNLOAD_POS_START_REQ
                   #sShuttleStartReq := NOT #iShuttleExtLoadUnloadAutoPos;
                   #sShuttlePosSetPoint := LREAL_TO_REAL(#iShuttleExtLoadUnloadAutoPosSetPoint);
                   #sCheck_Step_Condition := TRUE;
               END_REGION
           #S30_SHUTTLE_TO_EXT_LOAD_UNLOAD_POS_REACHED:
               REGION S30_SHUTTLE_TO_EXT_LOAD_UNLOAD_POS_REACHED
                   #sCheck_Step_Condition := TRUE;
               END_REGION
           #S40_SET_EXCHANGE_EXT_LOADER_LOAD_UNLOAD:
               REGION S40_SET_EXCHANGE_EXT_LOADER_LOAD_UNLOAD
                   #oStartCommunicationWithExtLoader := TRUE;
                   #sCheck_Step_Condition := TRUE;
               END_REGION
           #S50_EXCHANGE_EXT_LOADER_IN_PROGRESS:
               REGION S50_EXCHANGE_EXT_LOADER_IN_PROGRESS
                   #sCheck_Step_Condition := TRUE;
               END_REGION
           #S60_EXCHANGE_EXT_LOADER_ACQUIT:
               REGION S60_EXCHANGE_EXT_LOADER_ACQUIT
                   #oStartCommunicationWithExtLoader := FALSE;
                   #sCheck_Step_Condition := TRUE;
               END_REGION
           #S70_SET_EXCHANGE_EXT_LOADER_UNLOAD:
               REGION S70_SET_EXCHANGE_EXT_LOADER_UNLOAD
                   #oStartCommunicationWithExtLoader := TRUE;
                   #sCheck_Step_Condition := TRUE;
               END_REGION
           #S80_EXCHANGE_EXT_LOADER_IN_PROGRESS:
               REGION S80_EXCHANGE_EXT_LOADER_IN_PROGRESS
                   #sCheck_Step_Condition := TRUE;
               END_REGION
           #S90_EXCHANGE_EXT_LOADER_ACQUIT:
               REGION S90_EXCHANGE_EXT_LOADER_ACQUIT
                   #oStartCommunicationWithExtLoader := FALSE;
                   #sCheck_Step_Condition := TRUE;
               END_REGION
           #S100_SET_EXCHANGE_EXT_LOADER_UNLOAD:
               REGION S100_SET_EXCHANGE_EXT_LOADER_UNLOAD
                   #oStartCommunicationWithExtLoader := TRUE;
                   #sCheck_Step_Condition := TRUE;
               END_REGION
           #S110_EXCHANGE_EXT_LOADER_IN_PROGRESS:
               REGION S110_EXCHANGE_EXT_LOADER_IN_PROGRESS
                   #sCheck_Step_Condition := TRUE;
               END_REGION
           #S120_EXCHANGE_EXT_LOADER_ACQUIT:
               REGION S120_EXCHANGE_EXT_LOADER_ACQUIT
                   #oStartCommunicationWithExtLoader := FALSE;
                   #sCheck_Step_Condition := TRUE;
               END_REGION
           #S130_SHUTTLE_TO_EXT_LOAD_UNLOAD_MANU_POS_START_REQ:
               REGION S130_SHUTTLE_TO_EXT_LOAD_UNLOAD_MANU_POS_START_REQ
                   #sShuttleStartReq := NOT #iShuttleExtLoadUnloadManuPos;
                   #sShuttlePosSetPoint := LREAL_TO_REAL(#iShuttleExtLoadUnloadManuPosSetPoint);
                   #sCheck_Step_Condition := TRUE;
               END_REGION
           #S140_SHUTTLE_TO_EXT_LOAD_UNLOAD_MANU_POS_REACHED:
               REGION S140_SHUTTLE_TO_EXT_LOAD_UNLOAD_MANU_POS_REACHED
                   #sCheck_Step_Condition := TRUE;
               END_REGION
           #S150_OPERATOR_MESSAGE:
               REGION S150_OPERATOR_MESSAGE
                   #oSetLoadUnloadMsgManuMode := TRUE;
                   #sCheck_Step_Condition := TRUE;
               END_REGION
           #S195_JOB_DONE:
               REGION S95_JOB_DONE
                   #sInterface.JobDone := TRUE;
                   #sCheck_Step_Condition := TRUE;
               END_REGION
           ELSE:
               #sInterface.Error := TRUE;
       END_CASE;
   END_REGION

   REGION Sequence Next Step Condition
       IF #sCheck_Step_Condition THEN
           CASE #sCurrent_Step_NB OF
               #S00_INIT:
                   REGION S00 INIT
                       IF #sInterface.SequenceReleased AND #iJobReq THEN
                           #sCurrent_Step_NB := #S10_CHECK_EXT_LOAD_UNLOAD_OPTION;
                           #sInterface.SequenceRun := TRUE;
                           #sCheck_Step_Condition := FALSE;
                       ELSE
                           #sInterface.SequenceRun := FALSE;
                       END_IF;
                   END_REGION
               #S10_CHECK_EXT_LOAD_UNLOAD_OPTION:
                   REGION S10_CHECK_EXT_LOAD_UNLOAD_OPTION
                       IF #sInterface.SequenceReleased AND #sStepForward AND "DB_LoaderOptions".ExtLoadUnload.CommonPos AND #iAutoMode THEN
                           #sCurrent_Step_NB := #S20_SHUTTLE_TO_EXT_LOAD_UNLOAD_POS_START_REQ;
                           #sCheck_Step_Condition := FALSE;
                       ELSIF #sInterface.SequenceReleased AND #sStepForward AND #iSemiAutoMode THEN
                           #sCurrent_Step_NB := #S130_SHUTTLE_TO_EXT_LOAD_UNLOAD_MANU_POS_START_REQ;
                           #sCheck_Step_Condition := FALSE;
                       END_IF;
                   END_REGION
               #S20_SHUTTLE_TO_EXT_LOAD_UNLOAD_POS_START_REQ:
                   REGION S20_SHUTTLE_TO_EXT_LOAD_UNLOAD_POS_START_REQ
                       IF #sInterface.SequenceReleased AND (#iShuttleMoving OR #iShuttleExtLoadUnloadAutoPos) THEN
                           #sCurrent_Step_NB := #S30_SHUTTLE_TO_EXT_LOAD_UNLOAD_POS_REACHED;
                           #sCheck_Step_Condition := FALSE;
                       END_IF;
                   END_REGION
               #S30_SHUTTLE_TO_EXT_LOAD_UNLOAD_POS_REACHED:
                   REGION S30_SHUTTLE_TO_EXT_LOAD_UNLOAD_POS_REACHED
                       IF #sInterface.SequenceReleased AND #sStepForward AND NOT #sShuttleStartReq AND #iShuttleExtLoadUnloadAutoPos AND NOT #iEmptyingMode AND NOT #iFillingMode THEN
                           #sCurrent_Step_NB := #S40_SET_EXCHANGE_EXT_LOADER_LOAD_UNLOAD;
                           #sCheck_Step_Condition := FALSE;
                       ELSIF #sInterface.SequenceReleased AND #sStepForward AND NOT #sShuttleStartReq AND #iShuttleExtLoadUnloadAutoPos AND #iEmptyingMode AND NOT #iFillingMode THEN
                           #sCurrent_Step_NB := #S70_SET_EXCHANGE_EXT_LOADER_UNLOAD;
                           #sCheck_Step_Condition := FALSE;
                       ELSIF #sInterface.SequenceReleased AND #sStepForward AND NOT #sShuttleStartReq AND #iShuttleExtLoadUnloadAutoPos AND NOT #iEmptyingMode AND #iFillingMode THEN
                           #sCurrent_Step_NB := #S100_SET_EXCHANGE_EXT_LOADER_UNLOAD;
                           #sCheck_Step_Condition := FALSE;
                       END_IF;
                   END_REGION
               #S40_SET_EXCHANGE_EXT_LOADER_LOAD_UNLOAD:
                   REGION S40_SET_EXCHANGE_EXT_LOADER_LOAD_UNLOAD
                       IF #sInterface.SequenceReleased AND #sStepForward AND "AlwaysTRUE" THEN
                           #sCurrent_Step_NB := #S50_EXCHANGE_EXT_LOADER_IN_PROGRESS;
                           #sCheck_Step_Condition := FALSE;
                       END_IF;
                   END_REGION
               #S50_EXCHANGE_EXT_LOADER_IN_PROGRESS:
                   REGION S50_EXCHANGE_EXT_LOADER_IN_PROGRESS
                       IF #sInterface.SequenceReleased AND #sStepForward AND #iCommunicationWithExtLoaderDone THEN
                           #sCurrent_Step_NB := #S60_EXCHANGE_EXT_LOADER_ACQUIT;
                           #sCheck_Step_Condition := FALSE;
                       END_IF;
                   END_REGION
               #S60_EXCHANGE_EXT_LOADER_ACQUIT:
                   REGION S60_EXCHANGE_EXT_LOADER_ACQUIT
                       IF #sInterface.SequenceReleased AND #sStepForward AND "AlwaysTRUE" THEN
                           #sCurrent_Step_NB := #S195_JOB_DONE;
                           #sCheck_Step_Condition := FALSE;
                       END_IF;
                   END_REGION
               #S70_SET_EXCHANGE_EXT_LOADER_UNLOAD:
                   REGION S70_SET_EXCHANGE_EXT_LOADER_UNLOAD
                       IF #sInterface.SequenceReleased AND #sStepForward AND "AlwaysTRUE" THEN
                           #sCurrent_Step_NB := #S80_EXCHANGE_EXT_LOADER_IN_PROGRESS;
                           #sCheck_Step_Condition := FALSE;
                       END_IF;
                   END_REGION
               #S80_EXCHANGE_EXT_LOADER_IN_PROGRESS:
                   REGION S80_EXCHANGE_EXT_LOADER_IN_PROGRESS
                       IF #sInterface.SequenceReleased AND #sStepForward AND #iCommunicationWithExtLoaderDone THEN
                           #sCurrent_Step_NB := #S90_EXCHANGE_EXT_LOADER_ACQUIT;
                           #sCheck_Step_Condition := FALSE;
                       END_IF;
                   END_REGION
               #S90_EXCHANGE_EXT_LOADER_ACQUIT:
                   REGION S90_EXCHANGE_EXT_LOADER_ACQUIT
                       IF #sInterface.SequenceReleased AND #sStepForward AND "AlwaysTRUE" THEN
                           #sCurrent_Step_NB := #S195_JOB_DONE;
                           #sCheck_Step_Condition := FALSE;
                       END_IF;
                   END_REGION
               #S100_SET_EXCHANGE_EXT_LOADER_UNLOAD:
                   REGION S100_SET_EXCHANGE_EXT_LOADER_UNLOAD
                       IF #sInterface.SequenceReleased AND #sStepForward AND "AlwaysTRUE" THEN
                           #sCurrent_Step_NB := #S110_EXCHANGE_EXT_LOADER_IN_PROGRESS;
                           #sCheck_Step_Condition := FALSE;
                       END_IF;
                   END_REGION
               #S110_EXCHANGE_EXT_LOADER_IN_PROGRESS:
                   REGION S110_EXCHANGE_EXT_LOADER_IN_PROGRESS
                       IF #sInterface.SequenceReleased AND #sStepForward AND #iCommunicationWithExtLoaderDone THEN
                           #sCurrent_Step_NB := #S120_EXCHANGE_EXT_LOADER_ACQUIT;
                           #sCheck_Step_Condition := FALSE;
                       END_IF;
                   END_REGION
               #S120_EXCHANGE_EXT_LOADER_ACQUIT:
                   REGION S120_EXCHANGE_EXT_LOADER_ACQUIT
                       IF #sInterface.SequenceReleased AND #sStepForward AND "AlwaysTRUE" THEN
                           #sCurrent_Step_NB := #S195_JOB_DONE;
                           #sCheck_Step_Condition := FALSE;
                       END_IF;
                   END_REGION
               #S130_SHUTTLE_TO_EXT_LOAD_UNLOAD_MANU_POS_START_REQ:
                   REGION S130_SHUTTLE_TO_EXT_LOAD_UNLOAD_MANU_POS_START_REQ
                       IF #sInterface.SequenceReleased AND (#iShuttleMoving OR #iShuttleExtLoadUnloadManuPos) THEN
                           #sCurrent_Step_NB := #S140_SHUTTLE_TO_EXT_LOAD_UNLOAD_MANU_POS_REACHED;
                           #sCheck_Step_Condition := FALSE;
                       END_IF;
                   END_REGION
               #S140_SHUTTLE_TO_EXT_LOAD_UNLOAD_MANU_POS_REACHED:
                   REGION S140_SHUTTLE_TO_EXT_LOAD_UNLOAD_MANU_POS_REACHED
                       IF #sInterface.SequenceReleased AND #sStepForward AND NOT #sShuttleStartReq AND #iShuttleExtLoadUnloadManuPos THEN
                           #sCurrent_Step_NB := #S150_OPERATOR_MESSAGE;
                           #sCheck_Step_Condition := FALSE;
                       END_IF;
                   END_REGION
               #S150_OPERATOR_MESSAGE:
                   REGION S150_OPERATOR_MESSAGE
                       IF #sInterface.SequenceReleased AND #sStepForward AND #iLoadUnloadMsgManuModeAck THEN
                           #sCurrent_Step_NB := #S195_JOB_DONE;
                           #sCheck_Step_Condition := FALSE;
                       END_IF;
                   END_REGION
               #S195_JOB_DONE:
                   REGION S95_JOB_DONE
                       IF NOT #iJobReq THEN
                           #sCurrent_Step_NB := #S00_INIT;
                           #sCheck_Step_Condition := FALSE;
                           #sInterface.JobDone := FALSE;
                       END_IF;
                   END_REGION
               ELSE
                   #sInterface.Error := TRUE;
           END_CASE;
       END_IF;
   END_REGION

   REGION Outputs Update
       #oShuttleStartReq := #sShuttleStartReq;
       #oShuttlePosSetPoint := #sShuttlePosSetPoint;
   END_REGION

   REGION Steps - Date and Time History
       IF #sHistory.Activation THEN
           IF #sHistory.Steps[0] <> #sCurrent_Step_NB THEN
               FOR #tIndex := 98 TO 0 BY -1 DO
                   #sHistory.Steps[#tIndex + 1] := #sHistory.Steps[#tIndex];
                   #sHistory.Date_Time[#tIndex + 1] := #sHistory.Date_Time[#tIndex];
               END_FOR;
               #sHistory.Steps[0] := #sCurrent_Step_NB;
               #sHistory.Date_Time[0] := #iPLC_DateAndTime;
           END_IF;
       END_IF;
   END_REGION

   REGION Steps Text
       #StepText(iErrorCode := #sCurrent_Step_NB,
                 oErrorText => #StepText.oErrorText);
   END_REGION
END_FUNCTION_BLOCK

FUNCTION_BLOCK "FB_IntLoadUnload"   // FB62, SCL
{ S7_Optimized_Access := 'TRUE' }
// stored: AutoNumber false, MemoryReserve 100, SetENOAutomatically false
   VAR_INPUT
      iStartSeqCond : Bool;   // Start Sequence Conditions
      iJobReq : Bool;   // Job Request - From Main
      iShuttleIntLoadUnloadPos : Bool;   // Load/Unload Pos. Reached - Param
      iShuttleIntLoadUnloadPosSetPoint : LReal;   // Load/Unload Pos. Setpoint - Param
      iAxisV_LoadUnloadShuttlePos : Bool;
      iAxisV_LoadUnloadShuttlePosSetPoint : LReal;
      iAxisV_SafePos : Bool;
      iAxisV_SafePosSetPoint : LReal;
      iAxisW_SafePos : Bool;
      iAxisW_SafePosSetPoint : LReal;
      iAxisW_ApproachLoadUnloadPos : Bool;
      iAxisW_ApproachLoadUnloadSetPoint : LReal;
      iAxisW_LoadUnloadPos : Bool;
      iAxisW_LoadUnloadPosSetPoint : LReal;
      iShuttleMoving : Bool;   // Shuttle is moving - From FB_LoaderAxis
      iShuttleInPos : Bool;   // Shuttle pos. reached - From FB_LoaderAxis
      iAxisV_Moving : Bool;   // Shuttle is moving
      iAxisV_InPos : Bool;
      iAxisW_Moving { ExternalAccessible := 'False'; ExternalVisible := 'False'; ExternalWritable := 'False'} : Bool;   // Shuttle is moving
      iAxisW_InPos : Bool;
      iDrilledPartToUnload : Bool;   // Drilled Part To Unload - From FB_Position
      iUnDrilledPartToLoad : Bool;   // Unrilled Part To Load - From FB_Position
      iLoadGripperClosed : Bool;
      iUnloadGripperOpen : Bool;
      iPLC_DateAndTime : DTL;
      iStepPause : Bool;
   END_VAR
   VAR_OUTPUT
      oShuttleStartReq { ExternalAccessible := 'False'; ExternalVisible := 'False'; ExternalWritable := 'False'} : Bool;   // Shuttle Start Order - To FB_LoaderAxis
      oShuttlePosSetPoint { ExternalAccessible := 'False'; ExternalVisible := 'False'; ExternalWritable := 'False'} : Real;   // Shuttle Position Setpoint - To FB_LoaderAxis
      oAxisV_StartReq : Bool;
      oAxisV_PosSetPoint : Real;
      oAxisW_StartReq : Bool;
      oAxisW_PosSetPoint : Real;
      oLoadGripperCloseReq : Bool;
      oUnloadGripperOpenReq : Bool;
   END_VAR
   VAR
      sCurrent_Step_NB : Int;   // Active Step Number
      sCheck_Step_Condition : Bool;
      sOneStepForward : Bool;
      sRTOneStepForward : R_TRIG;
      sOneStepMode { S7_SetPoint := 'True'} : Bool;
      sStepForward : Bool;
      sInterface : "UDT_SequenceInterface";
      sShuttleStartReq { ExternalAccessible := 'False'; ExternalVisible := 'False'; ExternalWritable := 'False'} : Bool;
      sShuttlePosSetPoint { ExternalAccessible := 'False'; ExternalVisible := 'False'; ExternalWritable := 'False'} : Real;
      sAxisV_StartReq : Bool;
      sAxisV_PosSetPoint : Real;
      sAxisW_StartReq : Bool;
      sAxisW_PosSetPoint : Real;
      sLoadGripperCloseReq : Bool;   // Drilled Part To Unload - From FB_Position
      sUnloadGripperOpenReq : Bool;   // Unrilled Part To Load - From FB_Position
      sTimerAfterGripperClose : TON_TIME;
      sTimerAfterApproach { S7_SetPoint := 'True'} : TON_TIME;
      sHistory : Struct
         Activation : Bool;
         Steps : Array[0..99] of Int;
         Date_Time : Array[0..99] of DTL;
      END_STRUCT;
      StepText : "FB_GetTextErrorCode";
   END_VAR
   VAR_TEMP
      tIndex : Int;   // Index
   END_VAR
   VAR CONSTANT
      S00_INIT : Int := 0;
      S10_CHECK_INT_LOAD_UNLOAD_OPTION : Int := 10;
      S20_SHUTTLE_TO_INT_LOAD_UNLOAD_POS_START_REQ : Int := 20;
      S30_SHUTTLE_TO_INT_LOAD_UNLOAD_POS_REACHED : Int := 30;
      S40_AXIS_W_TO_SAFE_POS_START_REQ : Int := 40;
      S50_AXIS_W_TO_SAFE_POS_REACHED : Int := 50;
      S60_AXIS_V_TO_INT_LOAD_UNLOAD_POS_START_REQ : Int := 60;
      S70_AXIS_V_TO_INT_LOAD_UNLOAD_POS_REACHED : Int := 70;
      S80_AXIS_W_TO_INT_LOAD_UNLOAD_APPROACH_POS_START_REQ : Int := 80;
      S90_AXIS_W_TO_INT_LOAD_UNLOAD_APPROACH_POS_REACHED : Int := 90;
      S100_AXIS_W_TO_INT_LOAD_UNLOAD_POS_START_REQ : Int := 100;
      S110_AXIS_W_TO_INT_LOAD_UNLOAD_POS_REACHED : Int := 110;
      S120_OPEN_CLOSE_GRIPPER : Int := 120;
      S130_AXIS_W_TO_SAFE_POS_START_REQ : Int := 130;
      S140_AXIS_W_TO_SAFE_POS_REACHED : Int := 140;
      S150_AXIS_V_TO_SAFE_POS_START_REQ : Int := 150;
      S160_AXIS_V_TO_SAFE_POS_REACHED : Int := 160;
      S170_NO_PART_TO_LOAD_UNLOAD : Int := 170;
      S195_JOB_DONE : Int := 195;
   END_VAR
   // StepText.sCode_error[0].ErrorCode := 0;
   // StepText.sCode_error[1].ErrorCode := 10;
   // StepText.sCode_error[2].ErrorCode := 20;
   // StepText.sCode_error[3].ErrorCode := 30;
   // StepText.sCode_error[4].ErrorCode := 40;
   // StepText.sCode_error[5].ErrorCode := 50;
   // StepText.sCode_error[6].ErrorCode := 60;
   // StepText.sCode_error[7].ErrorCode := 70;
   // StepText.sCode_error[8].ErrorCode := 80;
   // StepText.sCode_error[9].ErrorCode := 90;
   // StepText.sCode_error[10].ErrorCode := 95;
BEGIN
   REGION Description header 
       //==================================================================================
       // POSALUX Swiss SA / (C) Copyright 2025
       //----------------------------------------------------------------------------------
       // Title: FB_ExtLoadUnload
       // Comment/Function: 
       // Author: Fabien WALDT
       // Engineering: TIA Portal v17
       //----------------------------------------------------------------------------------
       // Change log table:
       // Version  | Date     | Expert in charge | Changes applied
       // ---------|----------|------------------|-----------------------------------------
       // 00.00.01 | 20250527 | WFA              | First released version
       // =================================================================================
   END_REGION

   REGION Define condition to start
       IF #iStartSeqCond THEN
           #sInterface.SequenceReleased := TRUE;
       ELSE
           // Standard sequencer controls
           #sInterface.SequenceReleased := FALSE;
           #sCurrent_Step_NB := #S00_INIT;
           #sInterface.SequenceRun := FALSE;
           #sInterface.JobDone := FALSE;
           #sCheck_Step_Condition := FALSE;

           // Dedicated sequencer controls
           #sShuttleStartReq := FALSE;
           #sShuttlePosSetPoint := 0.0;
           #sAxisV_StartReq := FALSE;
           #sAxisV_PosSetPoint := 0.0;
           #sAxisW_StartReq := FALSE;
           #sAxisW_PosSetPoint := 0.0;
           #sLoadGripperCloseReq := FALSE;
           #sUnloadGripperOpenReq := FALSE;

           // Add specifics controls 
       END_IF;

       // Reset interface error
       IF #sInterface.Reset THEN
           #sInterface.Error := FALSE;
       END_IF;

       // Reset start when axis in position
       IF #iShuttleInPos THEN
           #sShuttleStartReq := FALSE;
       END_IF;
       IF #iAxisV_InPos THEN
           #sAxisV_StartReq := FALSE;
       END_IF;
       IF #iAxisW_InPos THEN
           #sAxisW_StartReq := FALSE;
       END_IF;

       // One step forward
       #sRTOneStepForward.CLK := #sOneStepForward;
       #sRTOneStepForward();
       #sStepForward := (NOT #sOneStepMode OR (#sOneStepMode AND #sRTOneStepForward.Q)) AND NOT #iStepPause;
       #sOneStepForward := FALSE;

       // Action only true in dedicated steps
       #sLoadGripperCloseReq := FALSE;
       #sUnloadGripperOpenReq := FALSE;

       // Timer Gripper OK
       #"sTimerAfterGripperClose"(IN := #sCurrent_Step_NB = 120
                                  AND(#iDrilledPartToUnload AND #iUnloadGripperOpen OR NOT #iDrilledPartToUnload)
                                  AND ((#iUnDrilledPartToLoad AND #iLoadGripperClosed) OR NOT #iUnDrilledPartToLoad),
                                  PT := T#500ms);

       // Timer between approach and Load/Unload position
       #sTimerAfterApproach(IN := #sCurrent_Step_NB = 90 AND #iAxisW_ApproachLoadUnloadPos,
                            PT := T#100ms);
   END_REGION

   REGION Sequence Function
       CASE #sCurrent_Step_NB OF
           #S00_INIT:
               REGION S00 INIT
                   #sCheck_Step_Condition := TRUE;
               END_REGION
           #S10_CHECK_INT_LOAD_UNLOAD_OPTION:
               REGION S10_CHECK_INT_LOAD_UNLOAD_OPTION
                   #sCheck_Step_Condition := TRUE;
               END_REGION
           #S20_SHUTTLE_TO_INT_LOAD_UNLOAD_POS_START_REQ:
               REGION S20_SHUTTLE_TO_INT_LOAD_UNLOAD_POS_START_REQ
                   #sShuttleStartReq := NOT #iShuttleIntLoadUnloadPos;
                   #sShuttlePosSetPoint := LREAL_TO_REAL(#iShuttleIntLoadUnloadPosSetPoint);
                   #sCheck_Step_Condition := TRUE;
               END_REGION
           #S30_SHUTTLE_TO_INT_LOAD_UNLOAD_POS_REACHED:
               REGION S30_SHUTTLE_TO_INT_LOAD_UNLOAD_POS_REACHED
                   #sCheck_Step_Condition := TRUE;
               END_REGION
           #S40_AXIS_W_TO_SAFE_POS_START_REQ:
               REGION S40_AXIS_W_TO_SAFE_POS_START_REQ
                   #sAxisW_StartReq := NOT #iAxisW_SafePos;
                   #sAxisW_PosSetPoint := LREAL_TO_REAL(#iAxisW_SafePosSetPoint);
                   #sCheck_Step_Condition := TRUE;
               END_REGION
           #S50_AXIS_W_TO_SAFE_POS_REACHED:
               REGION S50_AXIS_W_TO_SAFE_POS_REACHED
                   #sCheck_Step_Condition := TRUE;
               END_REGION
           #S60_AXIS_V_TO_INT_LOAD_UNLOAD_POS_START_REQ:
               REGION S60_AXIS_V_TO_INT_LOAD_UNLOAD_POS_START_REQ
                   #sAxisV_StartReq := NOT #iAxisV_LoadUnloadShuttlePos;
                   #sAxisV_PosSetPoint := LREAL_TO_REAL(#iAxisV_LoadUnloadShuttlePosSetPoint);
                       #sCheck_Step_Condition := TRUE;
                   END_REGION
           #S70_AXIS_V_TO_INT_LOAD_UNLOAD_POS_REACHED:
               REGION S70_AXIS_V_TO_INT_LOAD_UNLOAD_POS_REACHED
                   #sCheck_Step_Condition := TRUE;
               END_REGION
           #S80_AXIS_W_TO_INT_LOAD_UNLOAD_APPROACH_POS_START_REQ:
               REGION S80_AXIS_W_TO_INT_LOAD_UNLOAD_APPROACH_POS_START_REQ
                   #sAxisW_StartReq := NOT #iAxisW_ApproachLoadUnloadPos;
                   #sAxisW_PosSetPoint := LREAL_TO_REAL(#iAxisW_ApproachLoadUnloadSetPoint);
                   #sCheck_Step_Condition := TRUE;
               END_REGION
           #S90_AXIS_W_TO_INT_LOAD_UNLOAD_APPROACH_POS_REACHED:
               REGION S90_AXIS_W_TO_INT_LOAD_UNLOAD_APPROACH_POS_REACHED
                   IF #sTimerAfterApproach.Q THEN
                       #sCheck_Step_Condition := TRUE;
                   END_IF;
               END_REGION
           #S100_AXIS_W_TO_INT_LOAD_UNLOAD_POS_START_REQ:
               REGION S100_AXIS_W_TO_INT_LOAD_UNLOAD_POS_START_REQ
                   #sAxisW_StartReq := NOT #iAxisW_LoadUnloadPos;
                   #sAxisW_PosSetPoint := LREAL_TO_REAL(#iAxisW_LoadUnloadPosSetPoint);
                   #sCheck_Step_Condition := TRUE;
               END_REGION
           #S110_AXIS_W_TO_INT_LOAD_UNLOAD_POS_REACHED:
               REGION S110_AXIS_W_TO_INT_LOAD_UNLOAD_POS_REACHED
                   #sCheck_Step_Condition := TRUE;
               END_REGION
           #S120_OPEN_CLOSE_GRIPPER:
               REGION S120_OPEN_CLOSE_GRIPPER
                   #sLoadGripperCloseReq := #iUnDrilledPartToLoad;
                   #sUnloadGripperOpenReq := #iDrilledPartToUnload;
                   IF #"sTimerAfterGripperClose".Q THEN
                       #sCheck_Step_Condition := TRUE;
                   END_IF;
               END_REGION
           #S130_AXIS_W_TO_SAFE_POS_START_REQ:
               REGION S130_AXIS_W_TO_SAFE_POS_START_REQ
                   #sAxisW_StartReq := NOT #iAxisW_SafePos;
                   #sAxisW_PosSetPoint := LREAL_TO_REAL(#iAxisW_SafePosSetPoint);
                   #sCheck_Step_Condition := TRUE;
               END_REGION
           #S140_AXIS_W_TO_SAFE_POS_REACHED:
               REGION S140_AXIS_W_TO_SAFE_POS_REACHED
                   #sCheck_Step_Condition := TRUE;
               END_REGION
           #S150_AXIS_V_TO_SAFE_POS_START_REQ:
               REGION S150_AXIS_V_TO_SAFE_POS_START_REQ
                   #sAxisV_StartReq := NOT #iAxisV_SafePos;
                   #sAxisV_PosSetPoint := LREAL_TO_REAL(#iAxisV_SafePosSetPoint);
                   #sCheck_Step_Condition := TRUE;
               END_REGION
           #S160_AXIS_V_TO_SAFE_POS_REACHED:
               REGION S160_AXIS_V_TO_SAFE_POS_REACHED
                   #sCheck_Step_Condition := TRUE;
               END_REGION
           #S170_NO_PART_TO_LOAD_UNLOAD:
               REGION S170_NO_PART_TO_UNLOAD
                   #sCheck_Step_Condition := TRUE;
               END_REGION
           #S195_JOB_DONE:
               REGION S95_JOB_DONE
                   #sInterface.JobDone := TRUE;
                   #sCheck_Step_Condition := TRUE;
               END_REGION
           ELSE:
               #sInterface.Error := TRUE;
       END_CASE;
   END_REGION

   REGION Sequence Next Step Condition
       IF #sCheck_Step_Condition THEN
           CASE #sCurrent_Step_NB OF
               #S00_INIT:
                   REGION S00 INIT
                       IF #sInterface.SequenceReleased AND #iJobReq THEN
                           #sCurrent_Step_NB := #S10_CHECK_INT_LOAD_UNLOAD_OPTION;
                           #sInterface.SequenceRun := TRUE;
                           #sCheck_Step_Condition := FALSE;
                       ELSE
                           #sInterface.SequenceRun := FALSE;
                       END_IF;
                   END_REGION
               #S10_CHECK_INT_LOAD_UNLOAD_OPTION:
                   REGION S10_CHECK_INT_LOAD_UNLOAD_OPTION
                       IF #sInterface.SequenceReleased AND #sStepForward AND "DB_LoaderOptions".IntLoadUnload.CommonPos AND (#iDrilledPartToUnload OR #iUnDrilledPartToLoad) THEN
                           #sCurrent_Step_NB := #S20_SHUTTLE_TO_INT_LOAD_UNLOAD_POS_START_REQ;
                           #sCheck_Step_Condition := FALSE;
                       ELSIF #sInterface.SequenceReleased AND #sStepForward AND "DB_LoaderOptions".IntLoadUnload.CommonPos AND NOT #iJobReq OR (NOT #iDrilledPartToUnload AND NOT #iUnDrilledPartToLoad) THEN
                           #sCurrent_Step_NB := #S170_NO_PART_TO_LOAD_UNLOAD;
                           #sCheck_Step_Condition := FALSE;
                       END_IF;
                   END_REGION
               #S20_SHUTTLE_TO_INT_LOAD_UNLOAD_POS_START_REQ:
                   REGION S20_SHUTTLE_TO_INT_LOAD_UNLOAD_POS_START_REQ
                       IF #sInterface.SequenceReleased AND (#iShuttleMoving OR #iShuttleIntLoadUnloadPos) THEN
                           #sCurrent_Step_NB := #S30_SHUTTLE_TO_INT_LOAD_UNLOAD_POS_REACHED;
                           #sCheck_Step_Condition := FALSE;
                       END_IF;
                   END_REGION
               #S30_SHUTTLE_TO_INT_LOAD_UNLOAD_POS_REACHED:
                   REGION S30_SHUTTLE_TO_INT_LOAD_UNLOAD_POS_REACHED
                       IF #sInterface.SequenceReleased AND #sStepForward AND NOT #sShuttleStartReq AND #iShuttleIntLoadUnloadPos THEN
                           #sCurrent_Step_NB := #S60_AXIS_V_TO_INT_LOAD_UNLOAD_POS_START_REQ;
                           #sCheck_Step_Condition := FALSE;
                       END_IF;
                   END_REGION
               #S40_AXIS_W_TO_SAFE_POS_START_REQ:
                   REGION S40_AXIS_W_TO_SAFE_POS_START_REQ
                       IF #sInterface.SequenceReleased AND #sStepForward AND (#iAxisW_Moving OR #iAxisW_SafePos) THEN
                           #sCurrent_Step_NB := #S50_AXIS_W_TO_SAFE_POS_REACHED;
                           #sCheck_Step_Condition := FALSE;
                       END_IF;
                   END_REGION
               #S50_AXIS_W_TO_SAFE_POS_REACHED:
                   REGION S50_AXIS_W_TO_SAFE_POS_REACHED
                       IF #sInterface.SequenceReleased AND #sStepForward AND NOT #sAxisW_StartReq AND #iAxisW_SafePos THEN
                           #sCurrent_Step_NB := #S60_AXIS_V_TO_INT_LOAD_UNLOAD_POS_START_REQ;
                           #sCheck_Step_Condition := FALSE;
                       END_IF;
                   END_REGION
               #S60_AXIS_V_TO_INT_LOAD_UNLOAD_POS_START_REQ:
                   REGION S60_AXIS_V_TO_INT_LOAD_UNLOAD_POS_START_REQ
                       IF #sInterface.SequenceReleased AND (#iAxisV_Moving OR #iAxisV_LoadUnloadShuttlePos) THEN
                           #sCurrent_Step_NB := #S70_AXIS_V_TO_INT_LOAD_UNLOAD_POS_REACHED;
                           #sCheck_Step_Condition := FALSE;
                       END_IF;
                   END_REGION
               #S70_AXIS_V_TO_INT_LOAD_UNLOAD_POS_REACHED:
                   REGION S70_AXIS_V_TO_INT_LOAD_UNLOAD_POS_REACHED
                       IF #sInterface.SequenceReleased AND #sStepForward AND NOT #sAxisV_StartReq AND #iAxisV_LoadUnloadShuttlePos THEN
                           #sCurrent_Step_NB := #S80_AXIS_W_TO_INT_LOAD_UNLOAD_APPROACH_POS_START_REQ;
                           #sCheck_Step_Condition := FALSE;
                       END_IF;
                   END_REGION
               #S80_AXIS_W_TO_INT_LOAD_UNLOAD_APPROACH_POS_START_REQ:
                   REGION S80_AXIS_W_TO_INT_LOAD_UNLOAD_APPROACH_POS_START_REQ
                       IF #sInterface.SequenceReleased AND #sStepForward AND (#iAxisW_Moving OR #iAxisW_ApproachLoadUnloadPos) THEN
                           #sCurrent_Step_NB := #S90_AXIS_W_TO_INT_LOAD_UNLOAD_APPROACH_POS_REACHED;
                           #sCheck_Step_Condition := FALSE;
                       END_IF;
                   END_REGION
               #S90_AXIS_W_TO_INT_LOAD_UNLOAD_APPROACH_POS_REACHED:
                   REGION S90_AXIS_W_TO_INT_LOAD_UNLOAD_APPROACH_POS_REACHED
                       IF #sInterface.SequenceReleased AND #sStepForward AND NOT #sAxisW_StartReq AND #iAxisW_ApproachLoadUnloadPos THEN
                           #sCurrent_Step_NB := #S100_AXIS_W_TO_INT_LOAD_UNLOAD_POS_START_REQ;
                           #sCheck_Step_Condition := FALSE;
                       END_IF;
                   END_REGION
               #S100_AXIS_W_TO_INT_LOAD_UNLOAD_POS_START_REQ:
                   REGION S100_AXIS_W_TO_INT_LOAD_UNLOAD_POS_START_REQ
                       IF #sInterface.SequenceReleased AND (#iAxisW_Moving OR #iAxisW_LoadUnloadPos) THEN
                           #sCurrent_Step_NB := #S110_AXIS_W_TO_INT_LOAD_UNLOAD_POS_REACHED;
                           #sCheck_Step_Condition := FALSE;
                       END_IF;
                   END_REGION
               #S110_AXIS_W_TO_INT_LOAD_UNLOAD_POS_REACHED:
                   REGION S110_AXIS_W_TO_INT_LOAD_UNLOAD_POS_REACHED
                       IF #sInterface.SequenceReleased AND #sStepForward AND NOT #sAxisW_StartReq AND #iAxisW_LoadUnloadPos THEN
                           #sCurrent_Step_NB := #S120_OPEN_CLOSE_GRIPPER;
                           #sCheck_Step_Condition := FALSE;
                       END_IF;
                   END_REGION
               #S120_OPEN_CLOSE_GRIPPER:
                   REGION S120_OPEN_CLOSE_GRIPPER
                       IF #sInterface.SequenceReleased AND #sStepForward
                           AND (#iDrilledPartToUnload AND #iUnloadGripperOpen OR NOT #iDrilledPartToUnload)
                           AND ((#iUnDrilledPartToLoad AND #iLoadGripperClosed) OR NOT #iUnDrilledPartToLoad) THEN
                           #sCurrent_Step_NB := #S130_AXIS_W_TO_SAFE_POS_START_REQ;
                           #sCheck_Step_Condition := FALSE;
                       END_IF;
                   END_REGION
               #S130_AXIS_W_TO_SAFE_POS_START_REQ:
                   REGION S130_AXIS_W_TO_SAFE_POS_START_REQ
                       IF #sInterface.SequenceReleased AND (#iAxisW_Moving OR #iAxisW_SafePos) THEN
                           #sCurrent_Step_NB := #S140_AXIS_W_TO_SAFE_POS_REACHED;
                           #sCheck_Step_Condition := FALSE;
                       END_IF;
                   END_REGION
               #S140_AXIS_W_TO_SAFE_POS_REACHED:
                   REGION S140_AXIS_W_TO_SAFE_POS_REACHED
                       IF #sInterface.SequenceReleased AND #sStepForward AND NOT #sAxisW_StartReq AND #iAxisW_SafePos THEN
                         //  #sCurrent_Step_NB := #S150_AXIS_V_TO_SAFE_POS_START_REQ;
                           #sCurrent_Step_NB := #S195_JOB_DONE;
                           #sCheck_Step_Condition := FALSE;
                       END_IF;
                   END_REGION
               #S150_AXIS_V_TO_SAFE_POS_START_REQ:
                   REGION S150_AXIS_V_TO_SAFE_POS_START_REQ
                       IF #sInterface.SequenceReleased AND (#iAxisV_Moving OR #iAxisV_SafePos) THEN
                           #sCurrent_Step_NB := #S160_AXIS_V_TO_SAFE_POS_REACHED;
                           #sCheck_Step_Condition := FALSE;
                       END_IF;
                   END_REGION
               #S160_AXIS_V_TO_SAFE_POS_REACHED:
                   REGION S160_AXIS_V_TO_SAFE_POS_REACHED
                       IF #sInterface.SequenceReleased AND #sStepForward AND NOT #sAxisV_StartReq AND #iAxisV_SafePos THEN
                           #sCurrent_Step_NB := #S195_JOB_DONE;
                           #sCheck_Step_Condition := FALSE;
                       END_IF;
                   END_REGION
               #S170_NO_PART_TO_LOAD_UNLOAD:
                   REGION S170_NO_PART_TO_LOAD_UNLOAD
                       IF #sInterface.SequenceReleased AND #sStepForward AND "AlwaysTRUE" THEN
                           #sCurrent_Step_NB := #S130_AXIS_W_TO_SAFE_POS_START_REQ;
                           #sCheck_Step_Condition := FALSE;
                       END_IF;
                   END_REGION
               #S195_JOB_DONE:
                   REGION S195_JOB_DONE
                       IF NOT #iJobReq THEN
                           #sCurrent_Step_NB := #S00_INIT;
                           #sCheck_Step_Condition := FALSE;
                           #sInterface.JobDone := FALSE;
                       END_IF;
                   END_REGION
               ELSE
                   #sInterface.Error := TRUE;
           END_CASE;
       END_IF;
   END_REGION

   REGION Outputs Update
       #oShuttleStartReq := #sShuttleStartReq;
       #oShuttlePosSetPoint := #sShuttlePosSetPoint;
       #oAxisV_StartReq := #sAxisV_StartReq;
       #oAxisV_PosSetPoint := #sAxisV_PosSetPoint;
       #oAxisW_StartReq := #sAxisW_StartReq;
       #oAxisW_PosSetPoint := #sAxisW_PosSetPoint;
       #oLoadGripperCloseReq := #sLoadGripperCloseReq;
       #oUnloadGripperOpenReq := #sUnloadGripperOpenReq;

   END_REGION

   REGION Steps - Date and Time History
       IF #sHistory.Activation THEN
           IF #sHistory.Steps[0] <> #sCurrent_Step_NB THEN
               FOR #tIndex := 98 TO 0 BY -1 DO
                   #sHistory.Steps[#tIndex + 1] := #sHistory.Steps[#tIndex];
                   #sHistory.Date_Time[#tIndex + 1] := #sHistory.Date_Time[#tIndex];
               END_FOR;
               #sHistory.Steps[0] := #sCurrent_Step_NB;
               #sHistory.Date_Time[0] := #iPLC_DateAndTime;
           END_IF;
       END_IF;
   END_REGION

   REGION Steps Text
       #StepText(iErrorCode := #sCurrent_Step_NB,
                 oErrorText => #StepText.oErrorText);
   END_REGION
END_FUNCTION_BLOCK

FUNCTION_BLOCK "FB_IntLoadUnloadOP"   // FB73, SCL
{ S7_Optimized_Access := 'TRUE' }
// stored: AutoNumber false, MemoryReserve 100, SetENOAutomatically false
   VAR_INPUT
      iStartSeqCond : Bool;   // Start Sequence Conditions
      iJobReq : Bool;   // Job Request - From Main
      iShuttleIntLoadUnloadPos : Bool;   // Load/Unload Pos. Reached - Param
      iShuttleIntLoadUnloadPosSetPoint : LReal;   // Load/Unload Pos. Setpoint - Param
      iShuttleIntLoadUnloadOP_Pos : Bool;   // Load/Unload Pos. Reached - Param
      iShuttleIntLoadUnloadOP_PosSetPoint : LReal;   // Load/Unload Pos. Setpoint - Param
      iAxisV_LoadUnloadShuttlePos : Bool;
      iAxisV_LoadUnloadShuttlePosSetPoint : LReal;
      iAxisV_SafePos : Bool;
      iAxisV_SafePosSetPoint : LReal;
      iAxisW_SafePos : Bool;
      iAxisW_SafePosSetPoint : LReal;
      iAxisW_ApproachLoadUnloadPos : Bool;
      iAxisW_ApproachLoadUnloadSetPoint : LReal;
      iAxisW_LoadUnloadPos : Bool;
      iAxisW_LoadUnloadPosSetPoint : LReal;
      iShuttleMoving : Bool;   // Shuttle is moving - From FB_LoaderAxis
      iShuttleInPos : Bool;   // Shuttle pos. reached - From FB_LoaderAxis
      iAxisV_Moving : Bool;   // Shuttle is moving
      iAxisV_InPos : Bool;
      iAxisW_Moving { ExternalAccessible := 'False'; ExternalVisible := 'False'; ExternalWritable := 'False'} : Bool;   // Shuttle is moving
      iAxisW_InPos : Bool;
      iDrilledPartToUnload : Bool;   // Drilled Part To Unload - From FB_Position
      iUnDrilledPartToLoad : Bool;   // Unrilled Part To Load - From FB_Position
      iLoadGripperClosed : Bool;
      iUnloadGripperOpen : Bool;
      iPLC_DateAndTime : DTL;
      iStepPause : Bool;
   END_VAR
   VAR_OUTPUT
      oShuttleStartReq { ExternalAccessible := 'False'; ExternalVisible := 'False'; ExternalWritable := 'False'} : Bool;   // Shuttle Start Order - To FB_LoaderAxis
      oShuttlePosSetPoint { ExternalAccessible := 'False'; ExternalVisible := 'False'; ExternalWritable := 'False'} : Real;   // Shuttle Position Setpoint - To FB_LoaderAxis
      oAxisV_StartReq : Bool;
      oAxisV_PosSetPoint : Real;
      oAxisW_StartReq : Bool;
      oAxisW_PosSetPoint : Real;
      oLoadGripperCloseReq : Bool;
      oUnloadGripperOpenReq : Bool;
   END_VAR
   VAR
      sCurrent_Step_NB : Int;   // Active Step Number
      sCheck_Step_Condition : Bool;
      sOneStepForward : Bool;
      sRTOneStepForward : R_TRIG;
      sOneStepMode { S7_SetPoint := 'True'} : Bool;
      sStepForward : Bool;
      sInterface : "UDT_SequenceInterface";
      sShuttleStartReq { ExternalAccessible := 'False'; ExternalVisible := 'False'; ExternalWritable := 'False'} : Bool;
      sShuttlePosSetPoint { ExternalAccessible := 'False'; ExternalVisible := 'False'; ExternalWritable := 'False'} : Real;
      sAxisV_StartReq : Bool;
      sAxisV_PosSetPoint : Real;
      sAxisW_StartReq : Bool;
      sAxisW_PosSetPoint : Real;
      sLoadGripperCloseReq : Bool;   // Drilled Part To Unload - From FB_Position
      sUnloadGripperOpenReq : Bool;   // Unrilled Part To Load - From FB_Position
      sTimerAfterGripperClose : TON_TIME;
      sTimerAfterGripperOpen : TON_TIME;
      sTimerAfterApproach { S7_SetPoint := 'True'} : TON_TIME;
      sHistory : Struct
         Activation : Bool;
         Steps : Array[0..99] of Int;
         Date_Time : Array[0..99] of DTL;
      END_STRUCT;
      StepText : "FB_GetTextErrorCode";
   END_VAR
   VAR_TEMP
      tIndex : Int;   // Index
   END_VAR
   VAR CONSTANT
      S00_INIT : Int := 0;
      S10_CHECK_INT_LOAD_UNLOAD_OPTION : Int := 10;
      S20_SHUTTLE_TO_INT_LOAD_UNLOAD_POS_START_REQ : Int := 20;
      S30_SHUTTLE_TO_INT_LOAD_UNLOAD_POS_REACHED : Int := 30;
      S40_AXIS_W_TO_SAFE_POS_START_REQ : Int := 40;
      S50_AXIS_W_TO_SAFE_POS_REACHED : Int := 50;
      S60_AXIS_V_TO_INT_LOAD_UNLOAD_POS_START_REQ : Int := 60;
      S70_AXIS_V_TO_INT_LOAD_UNLOAD_POS_REACHED : Int := 70;
      S80_AXIS_W_TO_INT_LOAD_UNLOAD_APPROACH_POS_START_REQ : Int := 80;
      S90_AXIS_W_TO_INT_LOAD_UNLOAD_APPROACH_POS_REACHED : Int := 90;
      S100_AXIS_W_TO_INT_LOAD_UNLOAD_POS_START_REQ : Int := 100;
      S110_AXIS_W_TO_INT_LOAD_UNLOAD_POS_REACHED : Int := 110;
      S120_CLOSE_LOAD_GRIPPER : Int := 120;
      S130_AXIS_W_TO_SAFE_POS_START_REQ : Int := 130;
      S140_AXIS_W_TO_SAFE_POS_REACHED : Int := 140;
      S150_SHUTTLE_TO_INT_LOAD_UNLOAD_OP_POS_START_REQ : Int := 150;
      S160_SHUTTLE_TO_INT_LOAD_UNLOAD_OP_POS_REACHED : Int := 160;
      S170_AXIS_W_TO_INT_LOAD_UNLOAD_APPROACH_POS_START_REQ : Int := 170;
      S180_AXIS_W_TO_INT_LOAD_UNLOAD_APPROACH_POS_REACHED : Int := 180;
      S190_AXIS_W_TO_INT_LOAD_UNLOAD_POS_START_REQ : Int := 190;
      S200_AXIS_W_TO_INT_LOAD_UNLOAD_POS_REACHED : Int := 200;
      S210_OPEN_UNLOAD_GRIPPER : Int := 210;
      S220_AXIS_W_TO_SAFE_POS_START_REQ : Int := 220;
      S230_AXIS_W_TO_SAFE_POS_REACHED : Int := 230;
      S240_AXIS_V_TO_SAFE_POS_START_REQ : Int := 240;
      S250_AXIS_V_TO_SAFE_POS_REACHED : Int := 250;
      S260_NO_PART_TO_LOAD_UNLOAD : Int := 260;
      S295_JOB_DONE : Int := 295;
   END_VAR
   // StepText.sCode_error[0].ErrorCode := 0;
   // StepText.sCode_error[1].ErrorCode := 10;
   // StepText.sCode_error[2].ErrorCode := 20;
   // StepText.sCode_error[3].ErrorCode := 30;
   // StepText.sCode_error[4].ErrorCode := 40;
   // StepText.sCode_error[5].ErrorCode := 50;
   // StepText.sCode_error[6].ErrorCode := 60;
   // StepText.sCode_error[7].ErrorCode := 70;
   // StepText.sCode_error[8].ErrorCode := 80;
   // StepText.sCode_error[9].ErrorCode := 90;
   // StepText.sCode_error[10].ErrorCode := 95;
BEGIN
   REGION Description header 
       //==================================================================================
       // POSALUX Swiss SA / (C) Copyright 2026
       //----------------------------------------------------------------------------------
       // Title: FB_ExtLoadUnload_OP
       // Comment/Function: 
       // Author: Fabien WALDT
       // Engineering: TIA Portal v20
       //----------------------------------------------------------------------------------
       // Change log table:
       // Version  | Date     | Expert in charge | Changes applied
       // ---------|----------|------------------|-----------------------------------------
       // 00.00.01 | 20260128 | WFA              | First released version
       // =================================================================================
   END_REGION

   REGION Define condition to start
       IF #iStartSeqCond THEN
           #sInterface.SequenceReleased := TRUE;
       ELSE
           // Standard sequencer controls
           #sInterface.SequenceReleased := FALSE;
           #sCurrent_Step_NB := #S00_INIT;
           #sInterface.SequenceRun := FALSE;
           #sInterface.JobDone := FALSE;
           #sCheck_Step_Condition := FALSE;

           // Dedicated sequencer controls
           #sShuttleStartReq := FALSE;
           #sShuttlePosSetPoint := 0.0;
           #sAxisV_StartReq := FALSE;
           #sAxisV_PosSetPoint := 0.0;
           #sAxisW_StartReq := FALSE;
           #sAxisW_PosSetPoint := 0.0;
           #sLoadGripperCloseReq := FALSE;
           #sUnloadGripperOpenReq := FALSE;

           // Add specifics controls 
       END_IF;

       // Reset interface error
       IF #sInterface.Reset THEN
           #sInterface.Error := FALSE;
       END_IF;

       // Reset start when axis in position
       IF #iShuttleInPos THEN
           #sShuttleStartReq := FALSE;
       END_IF;
       IF #iAxisV_InPos THEN
           #sAxisV_StartReq := FALSE;
       END_IF;
       IF #iAxisW_InPos THEN
           #sAxisW_StartReq := FALSE;
       END_IF;

       // One step forward
       #sRTOneStepForward.CLK := #sOneStepForward;
       #sRTOneStepForward();
       #sStepForward := (NOT #sOneStepMode OR (#sOneStepMode AND #sRTOneStepForward.Q)) AND NOT #iStepPause;
       #sOneStepForward := FALSE;

       // Action only true in dedicated steps
       #sLoadGripperCloseReq := FALSE;
       #sUnloadGripperOpenReq := FALSE;

       // Timer Gripper OK
       #"sTimerAfterGripperClose"(IN := #sCurrent_Step_NB = 120
                                  AND ((#iUnDrilledPartToLoad AND #iLoadGripperClosed) OR NOT #iUnDrilledPartToLoad),
                                  PT := T#500ms);
       #"sTimerAfterGripperOpen"(IN := #sCurrent_Step_NB = 210
                                 AND ((#iDrilledPartToUnload AND #iUnloadGripperOpen) OR NOT #iDrilledPartToUnload),
                                 PT := T#500ms);

       // Timer between approach and Load/Unload position
       #sTimerAfterApproach(IN := (#sCurrent_Step_NB = 90 OR #sCurrent_Step_NB = 180) AND #iAxisW_ApproachLoadUnloadPos,
                            PT := T#100ms);
   END_REGION

   REGION Sequence Function
       CASE #sCurrent_Step_NB OF
           #S00_INIT:
               REGION S00 INIT
                   #sCheck_Step_Condition := TRUE;
               END_REGION
           #S10_CHECK_INT_LOAD_UNLOAD_OPTION:
               REGION S10_CHECK_INT_LOAD_UNLOAD_OPTION
                   #sCheck_Step_Condition := TRUE;
               END_REGION
           #S20_SHUTTLE_TO_INT_LOAD_UNLOAD_POS_START_REQ:
               REGION S20_SHUTTLE_TO_INT_LOAD_UNLOAD_POS_START_REQ
                   #sShuttleStartReq := NOT #iShuttleIntLoadUnloadPos;
                   #sShuttlePosSetPoint := LREAL_TO_REAL(#iShuttleIntLoadUnloadPosSetPoint);
                   #sCheck_Step_Condition := TRUE;
               END_REGION
           #S30_SHUTTLE_TO_INT_LOAD_UNLOAD_POS_REACHED:
               REGION S30_SHUTTLE_TO_INT_LOAD_UNLOAD_POS_REACHED
                   #sCheck_Step_Condition := TRUE;
               END_REGION
           #S40_AXIS_W_TO_SAFE_POS_START_REQ:
               REGION S40_AXIS_W_TO_SAFE_POS_START_REQ
                   #sAxisW_StartReq := NOT #iAxisW_SafePos;
                   #sAxisW_PosSetPoint := LREAL_TO_REAL(#iAxisW_SafePosSetPoint);
                   #sCheck_Step_Condition := TRUE;
               END_REGION
           #S50_AXIS_W_TO_SAFE_POS_REACHED:
               REGION S50_AXIS_W_TO_SAFE_POS_REACHED
                   #sCheck_Step_Condition := TRUE;
               END_REGION
           #S60_AXIS_V_TO_INT_LOAD_UNLOAD_POS_START_REQ:
               REGION S60_AXIS_V_TO_INT_LOAD_UNLOAD_POS_START_REQ
                   #sAxisV_StartReq := NOT #iAxisV_LoadUnloadShuttlePos;
                   #sAxisV_PosSetPoint := LREAL_TO_REAL(#iAxisV_LoadUnloadShuttlePosSetPoint);
                       #sCheck_Step_Condition := TRUE;
                   END_REGION
           #S70_AXIS_V_TO_INT_LOAD_UNLOAD_POS_REACHED:
               REGION S70_AXIS_V_TO_INT_LOAD_UNLOAD_POS_REACHED
                   #sCheck_Step_Condition := TRUE;
               END_REGION
           #S80_AXIS_W_TO_INT_LOAD_UNLOAD_APPROACH_POS_START_REQ:
               REGION S80_AXIS_W_TO_INT_LOAD_UNLOAD_APPROACH_POS_START_REQ
                   #sAxisW_StartReq := NOT #iAxisW_ApproachLoadUnloadPos;
                   #sAxisW_PosSetPoint := LREAL_TO_REAL(#iAxisW_ApproachLoadUnloadSetPoint);
                   #sCheck_Step_Condition := TRUE;
               END_REGION
           #S90_AXIS_W_TO_INT_LOAD_UNLOAD_APPROACH_POS_REACHED:
               REGION S90_AXIS_W_TO_INT_LOAD_UNLOAD_APPROACH_POS_REACHED
                   IF #sTimerAfterApproach.Q THEN
                       #sCheck_Step_Condition := TRUE;
                   END_IF;
               END_REGION
           #S100_AXIS_W_TO_INT_LOAD_UNLOAD_POS_START_REQ:
               REGION S100_AXIS_W_TO_INT_LOAD_UNLOAD_POS_START_REQ
                   #sAxisW_StartReq := NOT #iAxisW_LoadUnloadPos;
                   #sAxisW_PosSetPoint := LREAL_TO_REAL(#iAxisW_LoadUnloadPosSetPoint);
                   #sCheck_Step_Condition := TRUE;
               END_REGION
           #S110_AXIS_W_TO_INT_LOAD_UNLOAD_POS_REACHED:
               REGION S110_AXIS_W_TO_INT_LOAD_UNLOAD_POS_REACHED
                   #sCheck_Step_Condition := TRUE;
               END_REGION
           #S120_CLOSE_LOAD_GRIPPER:
               REGION S120_CLOSE_LOAD_GRIPPER
                   #sLoadGripperCloseReq := #iUnDrilledPartToLoad;
                   IF #"sTimerAfterGripperClose".Q THEN
                       #sCheck_Step_Condition := TRUE;
                   END_IF;
               END_REGION
           #S130_AXIS_W_TO_SAFE_POS_START_REQ:
               REGION S130_AXIS_W_TO_SAFE_POS_START_REQ
                   #sAxisW_StartReq := NOT #iAxisW_SafePos;
                   #sAxisW_PosSetPoint := LREAL_TO_REAL(#iAxisW_SafePosSetPoint);
                   #sCheck_Step_Condition := TRUE;
               END_REGION
           #S140_AXIS_W_TO_SAFE_POS_REACHED:
               REGION S140_AXIS_W_TO_SAFE_POS_REACHED
                   #sCheck_Step_Condition := TRUE;
               END_REGION
           #S150_SHUTTLE_TO_INT_LOAD_UNLOAD_OP_POS_START_REQ:
               REGION S150_SHUTTLE_TO_INT_LOAD_UNLOAD_OP_POS_START_REQ
                   #sShuttleStartReq := NOT #iShuttleIntLoadUnloadOP_Pos;
                   #sShuttlePosSetPoint := LREAL_TO_REAL(#iShuttleIntLoadUnloadOP_PosSetPoint);
                   #sCheck_Step_Condition := TRUE;
               END_REGION
           #S160_SHUTTLE_TO_INT_LOAD_UNLOAD_OP_POS_REACHED:
               REGION S160_SHUTTLE_TO_INT_LOAD_UNLOAD_OP_POS_REACHED
                   #sCheck_Step_Condition := TRUE;
               END_REGION
           #S170_AXIS_W_TO_INT_LOAD_UNLOAD_APPROACH_POS_START_REQ:
               REGION S170_AXIS_W_TO_INT_LOAD_UNLOAD_APPROACH_POS_START_REQ
                   #sAxisW_StartReq := NOT #iAxisW_ApproachLoadUnloadPos;
                   #sAxisW_PosSetPoint := LREAL_TO_REAL(#iAxisW_ApproachLoadUnloadSetPoint);
                   #sCheck_Step_Condition := TRUE;
               END_REGION
           #S180_AXIS_W_TO_INT_LOAD_UNLOAD_APPROACH_POS_REACHED:
               REGION S180_AXIS_W_TO_INT_LOAD_UNLOAD_APPROACH_POS_REACHED
                   IF #sTimerAfterApproach.Q THEN
                       #sCheck_Step_Condition := TRUE;
                   END_IF;
               END_REGION
           #S190_AXIS_W_TO_INT_LOAD_UNLOAD_POS_START_REQ:
               REGION S190_AXIS_W_TO_INT_LOAD_UNLOAD_POS_START_REQ
                   #sAxisW_StartReq := NOT #iAxisW_LoadUnloadPos;
                   #sAxisW_PosSetPoint := LREAL_TO_REAL(#iAxisW_LoadUnloadPosSetPoint);
                   #sCheck_Step_Condition := TRUE;
               END_REGION
           #S200_AXIS_W_TO_INT_LOAD_UNLOAD_POS_REACHED:
               REGION S200_AXIS_W_TO_INT_LOAD_UNLOAD_POS_REACHED
                   #sCheck_Step_Condition := TRUE;
               END_REGION
           #S210_OPEN_UNLOAD_GRIPPER:
               REGION S210_OPEN_UNLOAD_GRIPPER
                   #sUnloadGripperOpenReq := #iDrilledPartToUnload;
                   IF #"sTimerAfterGripperOpen".Q THEN
                       #sCheck_Step_Condition := TRUE;
                   END_IF;
               END_REGION
           #S220_AXIS_W_TO_SAFE_POS_START_REQ:
               REGION S220_AXIS_W_TO_SAFE_POS_START_REQ
                   #sAxisW_StartReq := NOT #iAxisW_SafePos;
                   #sAxisW_PosSetPoint := LREAL_TO_REAL(#iAxisW_SafePosSetPoint);
                   #sCheck_Step_Condition := TRUE;
               END_REGION
           #S230_AXIS_W_TO_SAFE_POS_REACHED:
               REGION S230_AXIS_W_TO_SAFE_POS_REACHED
                   #sCheck_Step_Condition := TRUE;
               END_REGION
           #S240_AXIS_V_TO_SAFE_POS_START_REQ:
               REGION S240_AXIS_V_TO_SAFE_POS_START_REQ
                   #sAxisV_StartReq := NOT #iAxisV_SafePos;
                   #sAxisV_PosSetPoint := LREAL_TO_REAL(#iAxisV_SafePosSetPoint);
                   #sCheck_Step_Condition := TRUE;
               END_REGION
           #S250_AXIS_V_TO_SAFE_POS_REACHED:
               REGION S250_AXIS_V_TO_SAFE_POS_REACHED
                   #sCheck_Step_Condition := TRUE;
               END_REGION
           #S260_NO_PART_TO_LOAD_UNLOAD:
               REGION S260_NO_PART_TO_LOAD_UNLOAD
                   #sCheck_Step_Condition := TRUE;
               END_REGION
           #S295_JOB_DONE:
               REGION S295_JOB_DONE
                   #sInterface.JobDone := TRUE;
                   #sCheck_Step_Condition := TRUE;
               END_REGION
           ELSE:
               #sInterface.Error := TRUE;
       END_CASE;
   END_REGION

